# B&R Automation Studio project TD52 (part 33)

### Module_ChargingUnit.var - Module global variables
```iecst
VAR
	bAMM_DPr_AirFilt_A_Hi : BOOL := FALSE; (*Warning charge air filter difference pressure high A*) (*V04.04.00.00*)
	bAMM_DPr_AirFilt_A_Lo : BOOL := FALSE; (*Warning charge air filter difference pressure low A*) (*V04.04.00.00*)
	bAMM_DPr_AirFilt_A_Ms : BOOL := FALSE; (*Warning measurement signal -  charge air filter difference pressure A*)
	bAMM_DPr_AirFilt_B_Hi : BOOL := FALSE; (*Warning charge air filter difference pressure high B*) (*V04.04.00.00*)
	bAMM_DPr_AirFilt_B_Lo : BOOL := FALSE; (*Warning charge air filter difference pressure low B*) (*V04.04.00.00*)
	bAMM_DPr_AirFilt_B_Ms : BOOL := FALSE; (*Warning measurement signal -  charge air filter difference pressure B*)
	bAMM_DPr_AirFilt_Hi : BOOL := FALSE; (*Warning charge air filter difference pressure high*) (*V04.04.00.00*)
	bAMM_DPr_AirFilt_Lo : BOOL := FALSE; (*Warning charge air filter difference pressure low*) (*V04.04.00.00*)
	bAMM_DPr_AirFilt_Ms : BOOL := FALSE; (*Warning measurement signal -  charge air filter difference pressure*)
	bAMM_DPr_Ch_FA_Hi : BOOL := FALSE; (*Warning difference pressure over flame arrester maximum*) (*V04.04.00.00*)
	bAMM_DPr_Ch_HPCooler_Hi : BOOL := FALSE; (*Warning difference pressure over high pressure charge cooler maximum*) (*V04.04.00.00*)
	bAMM_DPr_Ch_LPCooler_Hi : BOOL := FALSE; (*Warning difference pressure over  low pressure charge cooler maximum*) (*V04.04.00.00*)
	bAMM_DPr_Ch_P2s_Hi : BOOL := FALSE; (*Warning charge pressure p2' deviation maximum*) (*V04.07.00.00*)
	bAMM_DPr_Ch_P2s_HiHi : BOOL := FALSE; (*Error charge pressure p2' deviation maximum*)
	bAMM_DPr_Ch_P2_Hi : BOOL := FALSE; (*Warning charge pressure p2 deviation maximum*)
	bAMM_N_TCHP_A_Ms : BOOL := FALSE; (*Warning measurement signal - High pressure turbocharger speed A *)
	bAMM_N_TCHP_B_Ms : BOOL := FALSE; (*Warning measurement signal - High pressure turbocharger speed B*)
	bAMM_N_TCHP_Diff_Hi : BOOL := FALSE; (*Warning High pressure turbocharger speed deviation maximum*)
	bAMM_N_TCHP_Diff_HiHi : BOOL := FALSE; (*Error High pressure turbocharger speed deviation maximum*)
	bAMM_N_TCHP_Hi : BOOL := FALSE; (*Warning High pressure turbocharger speed maximum*)
	bAMM_N_TCHP_HiHi : BOOL := FALSE; (*Error High pressure turbocharger speed maximum*)
	bAMM_N_TCHP_Ms : BOOL := FALSE; (*Warning measurement signal - High pressure turbocharger speed *)
	bAMM_N_TCHP_MsMs : BOOL := FALSE; (*Error measurement signal - BOTH High pressure turbocharger speed *) (*V04.05.01.00*)
	bAMM_N_TCLP_A_Ms : BOOL := FALSE; (*Warning measurement signal - Low pressure turbocharger speed A *)
	bAMM_N_TCLP_B_Ms : BOOL := FALSE; (*Warning measurement signal - Low pressure turbocharger speed B*)
	bAMM_N_TCLP_Diff_Hi : BOOL := FALSE; (*Warning Low pressure turbocharger speed deviation maximum*)
	bAMM_N_TCLP_Diff_HiHi : BOOL := FALSE; (*Error Low pressure turbocharger speed deviation maximum*)
	bAMM_N_TCLP_Hi : BOOL := FALSE; (*Warning Low pressure turbocharger speed maximum*)
	bAMM_N_TCLP_HiHi : BOOL := FALSE; (*Error Low pressure turbocharger speed maximum*)
	bAMM_N_TCLP_Ms : BOOL := FALSE; (*Warning measurement signal - Low pressure turbocharger speed*)
	bAMM_N_TCLP_MsMs : BOOL := FALSE; (*Error measurement signal - BOTH Low pressure turbocharger speed*) (*V04.05.01.00*)
	bAMM_Pr_Ch_OoR : BOOL := FALSE; (*Warning for pressure signals out of range in standstill*)
	bAMM_Pr_Ch_P1HP_A_Ms : BOOL := FALSE; (*Warning measurement signal -  charge pressure p1 before high pressure TC A *)
	bAMM_Pr_Ch_P1HP_B_Ms : BOOL := FALSE; (*Warning measurement signal -  charge pressure p1 before high pressure TC A *)
	bAMM_Pr_Ch_P1HP_Ms : BOOL := FALSE; (*Warning measurement signal -  charge pressure p1 before high pressure TC *)
	bAMM_Pr_Ch_P1LP_A_Ms : BOOL := FALSE; (*Warning measurement signal - charge pressure before  low pressure turbocharger A*) (*V04.04.00.00*)
	bAMM_Pr_Ch_P1LP_B_Ms : BOOL := FALSE; (*Warning measurement signal - charge pressure before  low pressure turbocharger B*) (*V04.04.00.00*)
	bAMM_Pr_Ch_P2bFA_Ms : BOOL := FALSE; (*Warning measurement signal - charge pressure before flame arrester*) (*V04.04.00.00*)
	bAMM_Pr_Ch_P2HP_A_Ms : BOOL := FALSE; (*Warning measurement signal - charge pressure after high pressure turbocharger A*) (*V04.04.00.00*)
	bAMM_Pr_Ch_P2HP_B_Ms : BOOL := FALSE; (*Warning measurement signal - charge pressure after high pressure turbocharger B*) (*V04.04.00.00*)
	bAMM_Pr_Ch_P2HP_Ms : BOOL := FALSE; (*Warning measurement signal - charge pressure after high pressure turbocharger*) (*V04.04.00.00*)
	bAMM_Pr_Ch_P2LP_A_Ms : BOOL := FALSE; (*Warning measurement signal - charge pressure after  low pressure turbocharger A*) (*V04.04.00.00*)
	bAMM_Pr_Ch_P2LP_B_Ms : BOOL := FALSE; (*Warning measurement signal - charge pressure after  low pressure turbocharger B*) (*V04.04.00.00*)
	bAMM_Pr_Ch_P2LP_Ms : BOOL := FALSE; (*Warning measurement signal - charge pressure after  low pressure turbocharger*) (*V04.04.00.00*)
	bAMM_Pr_Ch_P2s_A_Ms : BOOL := FALSE; (*Warning measurement signal -  charge pressure p2' A *)
	bAMM_Pr_Ch_P2s_B_Ms : BOOL := FALSE; (*Warning measurement signal -  charge pressure p2' B*)
	bAMM_Pr_Ch_P2s_MsMs : BOOL := FALSE; (*Error measurement signal -  charge pressure p2' *)
	bAMM_Pr_Ch_P2_A_Ms : BOOL := FALSE; (*Warning measurement signal -  charge pressure p2 A*)
	bAMM_Pr_Ch_P2_B_Ms : BOOL := FALSE; (*Warning measurement signal -  charge pressure p2 B*)
	bAMM_Pr_Ch_P2_MsMs : BOOL := FALSE; (*Error measurement signal -  charge pressure p2 *)
	bAMM_Pr_Ch_P2_Sum_MsMs : BOOL := FALSE; (*Error measurement signal -  sum fault charge pressure *)
	bAMM_T_Ch_T1HP_A_Ms : BOOL := FALSE; (*Warning measurement signal -  charge temperature before high pressure TC  A*) (*V04.05.00.00*)
	bAMM_T_Ch_T1HP_B_Ms : BOOL := FALSE; (*Warning measurement signal -  charge temperature before high pressure TC  B*) (*V04.05.00.00*)
	bAMM_T_Ch_T1HP_Lo : BOOL := FALSE; (*Warning charge temperature before high pressure TC minimum*)
	bAMM_T_Ch_T1HP_MsMs : BOOL := FALSE; (*Error measurement signal -  charge temperature before high pressure TC  *)
	bAMM_T_Ch_T1LP_A_Ms : BOOL := FALSE; (*Warning measurement signal - charge temperature before turbocharger (air intake) A*) (*V04.04.00.00*)
	bAMM_T_Ch_T1LP_B_Ms : BOOL := FALSE; (*Warning measurement signal - charge temperature before turbocharger (air intake) B*) (*V04.04.00.00*)
	bAMM_T_Ch_T1LP_Ms : BOOL := FALSE; (*Warning measurement signal - charge temperature before turbocharger (air intake)*) (*V04.04.00.00*)
	bAMM_T_Ch_T2HP_A_Ms : BOOL := FALSE; (*Warning measurement signal -  charge temperature after high pressure TC  A*) (*V04.05.00.00*)
	bAMM_T_Ch_T2HP_B_Ms : BOOL := FALSE; (*Warning measurement signal -  charge temperature after high pressure TC  B*) (*V04.05.00.00*)
	bAMM_T_Ch_T2HP_HiHi : BOOL := FALSE; (*Error charge temperature after high pressure TC maximum*) (*V04.12.00.00*)
	bAMM_T_Ch_T2HP_Ms : BOOL := FALSE; (*Warning measurement signal -  charge temperature after high pressure TC *) (*V04.05.00.00*)
	bAMM_T_Ch_T2LP_A_Ms : BOOL := FALSE; (*Warning measurement signal -  charge temperature after low pressure TC  A*) (*V04.05.00.00*)
	bAMM_T_Ch_T2LP_B_Ms : BOOL := FALSE; (*Warning measurement signal -  charge temperature after low pressure TC  B*) (*V04.05.00.00*)
	bAMM_T_Ch_T2LP_HiHi : BOOL := FALSE; (*Error charge temperature after low pressure TC maximum*) (*V04.12.00.00*)
	bAMM_T_Ch_T2LP_Ms : BOOL := FALSE; (*Warning measurement signal -  charge temperature after low pressure TC *) (*V04.05.00.00*)
	bAMM_T_Ch_T2s_A_Hi : BOOL := FALSE; (*Warning charge temperature t2' A maximum*)
	bAMM_T_Ch_T2s_A_HiHi : BOOL := FALSE; (*Error charge temperature t2' A maximum*)
	bAMM_T_Ch_T2s_A_Lo : BOOL := FALSE; (*Warning charge temperature t2' A minimum*)
	bAMM_T_Ch_T2s_A_Ms : BOOL := FALSE; (*Warning measurement signal -  charge temperature t2' A*)
	bAMM_T_Ch_T2s_A_RocHiHi : BOOL := FALSE; (*Error charge temperature t2' A rate of change maximum*)
	bAMM_T_Ch_T2s_B_Hi : BOOL := FALSE; (*Warning charge temperature t2' B maximum*)
	bAMM_T_Ch_T2s_B_HiHi : BOOL := FALSE; (*Error charge temperature t2' B maximum*)
	bAMM_T_Ch_T2s_B_Lo : BOOL := FALSE; (*Warning charge temperature t2' B minimum*)
	bAMM_T_Ch_T2s_B_Ms : BOOL := FALSE; (*Warning measurement signal -  charge temperature t2' B*)
	bAMM_T_Ch_T2s_B_RocHiHi : BOOL := FALSE; (*Error charge temperature t2' B rate of change maximum*)
	bAMM_T_Ch_T2s_DiffHi : BOOL := FALSE; (*Warning charge temperature t2' inclination maximum*)
	bAMM_T_Ch_T2s_Hi : BOOL := FALSE; (*Warning charge temperature t2' maximum*)
	bAMM_T_Ch_T2s_HiHi : BOOL := FALSE; (*Error charge temperature t2' maximum*)
	bAMM_T_Ch_T2s_Lo : BOOL := FALSE; (*Warning charge temperature t2' minimum*)
	bAMM_T_Ch_T2s_MsMs : BOOL := FALSE; (*Error measurement signal -  charge temperature t2' *)
	bAMM_T_Ch_T2s_RocHiHi : BOOL := FALSE; (*Error charge temperature t2' rate of change maximum*)
	bAMM_T_Ch_T2_Calc : BOOL := FALSE; (*Warning intercooler inlet temperature not definable*) (*V04.12.00.00*)
	bGCB_On_300s : BOOL := FALSE; (*generator circuit breaker CLOSED + 300s*) (*V04.04.00.00*)
	bGnlTrip : BOOL; (*general alarm trip *)
	bGnlTrip1 : BOOL; (*general alarm trip priority 1*)
	bGnlTrip2 : BOOL; (*general alarm trip priority 2*)
	bGnlTrip3 : BOOL; (*general alarm trip priority 3*)
	bGnlWarning : BOOL; (*general alarm warning *)
	bNetP_Island_20s : BOOL := FALSE; (*Mains parallel operation mode or island mode for 20s*) (*V04.06.00.00*)
	bNoInitDetected : BOOL := FALSE; (*allways true, except 1cycle on init up*)
	bOMSS_MAT : BOOL; (*operation mode selector switch - MANUAL/AUTO/TEST*)
	bP_Nom10_60s : BOOL := FALSE; (*engine power >= 10% of nominal power for 60s*)
	bP_Nom10_300s : BOOL := FALSE; (*engine power >= 10% of nominal power for 300s*)
	bP_Nom10_600s : BOOL := FALSE; (*engine power >= 10% of nominal power for 600s*) (*V04.04.00.00*)
	bP_Nom50_30s : BOOL := FALSE; (*engine power >= 50% of nominal power for 30s*)
	bP_Nom75_02s : BOOL := FALSE; (*engine power >= 75% of nominal power for 2s*) (*V04.04.00.00*)
	bRelModul_ParaSetupOk : BOOL := FALSE; (*Release Module if ParaSetupOk = TRUE*) (*V04.04.00.00*)
	bRelModul_Sys_Run : BOOL := FALSE; (*Release Module if Sys_Run = TRUE*)
	bStartSpd : BOOL := FALSE; (*start speed reached*)
	gastype : INT := 0; (*Actual gas type*)
	iCnt_OpHours_LastCalib : DINT; (*Perm: Actual operating hours at time of calibration*) (*V04.04.00.00*)
	IN_CH : IN_CH_Struct; (*Module IN-Interface*)
	MM2VIS : MM2VIS_Struct; (*Module VISU-Interface (Module --> VISU)*)
	OUT_CH : OUT_CH_Struct; (*Module OUT-Interface*)
	Para : PARA_CH_Struct; (*Module Parameter-Interface*)
	ParaFactoryDefault : PARA_CH_Struct := (0); (*First Init Values*)
	pm : PARA_CH_Struct; (*Stored parameter structure *)
	rNum_Ch_CBV_Valve : REAL := 0.0; (*Number of compressor bypass valve *) (*V04.04.00.00*)
	rP_Act_LastCalib : REAL; (*Perm: Actual electric power at time of calibration [kW]*) (*V04.04.00.00*)
	rT_Ch_T1HP_Max : REAL; (*maximum value - charge temperature before high-pressure TC *) (*V04.05.01.00*)
	rT_Ch_T1LP_Max : REAL; (*maximum value - charge temperature before low-pressure TC *) (*V04.05.01.00*)
	rVol_Ch_AirFilt_Pnom : REAL; (*Perm: Extrapolated value for operation volume flow at nominal power [m³/h]*) (*V04.04.00.00*)
	xEngType : EngType; (*Instance of FB EngType*) (*V04.04.00.00*)
	xOpMode : OpMode := (0); (*Function block for operation mode*)
END_VAR
```

### Program Logical/ChargingUnit/GeneralCH (IEC, version 4.12.0) - general functions

#### GeneralCHCyclic.st - Cyclic code
```iecst
(*******************************************************************************
GeneralCH		general functions

This code is confidential and proprietary to the INNIO Company.
It may not be used in any form, or reproduced in any manner,
without the express written permission of the INNIO Company.
Copyright, INNIO Company, 2019

Customized modifications: -
------------------------

History:
-------
V03.99.00.00	18.03.2013 	Tinello 	Created
V04.04.00.00	18.05.2016 	Tinello 	bP_Nom10_600s added for Spec Vers. c
										Release Module, number of CBV and motor type added
										bP_Nom75_02s, bGCB_On_300s added
V04.06.00.00	01.10.2018 	Tinello 	bNetP_Island_20s added
V04.07.00.00	04.12.2018 	Tinello 	Number of compressor bypass valves added for engine type 4
V04.12.00.00	23.03.2023	Tinello		Added release Sys_Run

(*******************************************************************************)

PROGRAM _CYCLIC

	(* Release Module if ParaSetupOk = TRUE *)
	xTON_ParaSetupOk(IN		:= IN_CH.tPB2MM.bParaSetupOk, PT:= T#10s);
	bRelModul_ParaSetupOk	:= xTON_ParaSetupOk.Q;

	xTON_Sys_Run(IN			:= IN_CH.tPB2MM.bSys_Run, PT:= T#60s);
	bRelModul_Sys_Run		:= xTON_Sys_Run.Q;

	(* Engine motortype *)
	xEngType.Motortype 	:= INT_TO_UINT(Para.iEng_Motortype);
	xEngType();

	(* Operation mode selector switch *)
	bOMSS_MAT 	:= (IN_CH.iIdx_OMSS = 1) OR (IN_CH.iIdx_OMSS = 2) OR (IN_CH.iIdx_OMSS = 3);	(* 1= manual; 2= auto; 3= test mode *)

	(* engine start speed reached *)
	xGR_MAXR_StartSpd(In:= IN_CH.rN_EngAct, Gw := Para.rN_EngStart_LimHi, Hy := Para.rN_EngStart_HyHi);
	xTOF_StartSpd(IN 	:= xGR_MAXR_StartSpd.Q AND bRelModul_ParaSetupOk, PT := T#10s);
	bStartSpd			:= xTOF_StartSpd.Q;

	(* engine power > 10%Pn + 60s / 300s *)
	xGR_MAXR_P_Act10(In := IN_CH.rP_Act_Norm_Filt, Gw:= 0.1, Hy:= 0.01);
	xTON_P_Act10_60(IN	:= xGR_MAXR_P_Act10.Q AND bRelModul_ParaSetupOk AND IN_CH.tGCB_On.Di, PT:= T#60s);
	xTON_P_Act10_300(IN	:= xGR_MAXR_P_Act10.Q AND bRelModul_ParaSetupOk AND IN_CH.tGCB_On.Di, PT:= T#300s);
	xTON_P_Act10_600(IN	:= xGR_MAXR_P_Act10.Q AND bRelModul_ParaSetupOk AND IN_CH.tGCB_On.Di, PT:= T#600s);

	bP_Nom10_60s 		:= xTON_P_Act10_60.Q;
	bP_Nom10_300s 		:= xTON_P_Act10_300.Q;
	bP_Nom10_600s 		:= xTON_P_Act10_600.Q;

	(* engine power > 50%Pn + 30s *)
	xGR_MAXR_P_Act50(In := IN_CH.rP_Act_Norm_Filt, Gw:= 0.5, Hy:= 0.01);
	xTON_P_Act50_30(IN	:= xGR_MAXR_P_Act50.Q AND bRelModul_ParaSetupOk AND IN_CH.tGCB_On.Di, PT:= T#30s);

	bP_Nom50_30s 		:= xTON_P_Act50_30.Q;

	(* engine power > 75%Pn + 2s *)
	xGR_MAXR_P_Act75(In := IN_CH.rP_Act_Norm_Filt, Gw:= 0.75, Hy:= 0.05);
	xTON_P_Act75_02(IN	:= xGR_MAXR_P_Act75.Q AND bRelModul_ParaSetupOk AND IN_CH.tGCB_On.Di, PT:= T#2s);

	bP_Nom75_02s 		:= xTON_P_Act75_02.Q;

	(* generator circuit breaker CLOSED + 300s *)
	xTON_GCB_On_300(IN	:= IN_CH.tGCB_On.Di, PT:= T#300s);
	bGCB_On_300s 		:= xTON_GCB_On_300.Q;

	(* call function for the state machine - engine operation mode *)
	xOpMode(in 	:= IN_CH.iSt_OpMode);

	(* Mains parallel operation mode / island mode + 20s *)
	xTON_NetP_Island_20(IN	:= xOpMode.NetP OR xOpMode.Island, PT:= T#20s);
	bNetP_Island_20s		:= xTON_NetP_Island_20.Q;

	(* gastype *)
	gastype	:= IN_CH.iIdx_Gtyp_Dem;

	(* Number of compressor bypass valves *)
	CASE Para.iEng_Motortype OF
		412:	IF xOpMode.Island						 	THEN	rNum_Ch_CBV_Valve	:= 2;
															ELSE	rNum_Ch_CBV_Valve	:= 1;
				END_IF
		416:	IF xOpMode.Island						 	THEN	rNum_Ch_CBV_Valve	:= 2;
															ELSE	rNum_Ch_CBV_Valve	:= 1;
				END_IF
		420:	IF xOpMode.Island						 	THEN	rNum_Ch_CBV_Valve	:= 2;
															ELSE	rNum_Ch_CBV_Valve	:= 1;
				END_IF
		424:	IF xOpMode.Island						 	THEN	rNum_Ch_CBV_Valve	:= 2;
															ELSE	rNum_Ch_CBV_Valve	:= 1;
				END_IF
		612:														rNum_Ch_CBV_Valve	:= 1;
		616:														rNum_Ch_CBV_Valve	:= 2;
		620:														rNum_Ch_CBV_Valve	:= 3;
		624:	IF FIND(IN_CH.szEng_Motorversion, 'H') = 1 	THEN	rNum_Ch_CBV_Valve	:= 2;
															ELSE	rNum_Ch_CBV_Valve	:= 4;
				END_IF
		920:														rNum_Ch_CBV_Valve	:= 2;
	END_CASE

END_PROGRAM
```

#### GeneralCH.var - Local variables
```iecst
VAR
	xGR_MAXR_P_Act10 : GR_MAXR := (0); (*FuB*)
	xGR_MAXR_P_Act50 : GR_MAXR := (0); (*FuB*)
	xGR_MAXR_P_Act75 : GR_MAXR := (0); (*FuB*)
	xGR_MAXR_StartSpd : GR_MAXR := (0); (*Engine start speed passed*)
	xTOF_StartSpd : TOF := (0); (*FuB*)
	xTON_GCB_On_300 : TON := (0); (*FuB*)
	xTON_NetP_Island_20 : TON := (0); (*FuB*)
	xTON_ParaSetupOk : TON := (0); (*FuB*)
	xTON_P_Act10_60 : TON := (0); (*FuB*)
	xTON_P_Act10_300 : TON := (0); (*FuB*)
	xTON_P_Act10_600 : TON := (0); (*FuB*)
	xTON_P_Act50_30 : TON := (0); (*FuB*)
	xTON_P_Act75_02 : TON := (0); (*FuB*)
	xTON_Sys_Run : TON := (0); (*FuB*)
END_VAR
```

### Program Logical/ChargingUnit/DefaultCH (IEC, version 4.00.0) - Settings default values

#### DefaultCHCyclic.st - Cyclic code
```iecst
(*******************************************************************************
DefaultCH		value set

This code is confidential and proprietary to the INNIO Company.
It may not be used in any form, or reproduced in any manner,
without the express written permission of the INNIO Company.
Copyright, INNIO Company, 2019

Customized modifications: -
------------------------

History:
-------
V03.99.00.00	11.09.2012	Tinello		new

Instructions for use:
--------------------
- Default TRUE setting for not existing Di's

Outstandings:
------------

*******************************************************************************)
PROGRAM _CYCLIC

END_PROGRAM
```

### Program Logical/ChargingUnit/CH_SpeedTC (IEC, version 4.12.0) - turbo charger speed

#### CH_SpeedTCCyclic.st - Cyclic code
```iecst
(*******************************************************************************
TC_Speed	 		 turbocharger speed

This code is confidential and proprietary to the INNIO Company.
It may not be used in any form, or reproduced in any manner,
without written permission of the INNIO Company.
Copyright, INNIO Company, 2023

- turbocharger speed measuring
- speed and signal monitoring
- power reduction

Customized modifications: -
------------------------

History:
-------
V03.99.00.00	18.03.2013	Tinello		restructured
V04.00.00.00	01.09.2014	Tinello		If engine speed = 0 and no measurement failure -> TC speed is set to 0
V04.04.00.00	27.10.2016	Tinello		change of speed deviation function -> Spec.(b)
V04.05.00.00	23.01.2018	Tinello		Release Monitoring hinzu und Warnmanagement vereinfacht
V04.05.01.00	15.03.2018	Tinello		Spezifikation c
V04.05.03.00	28.05.2018	Tinello		Bugfix: Quittierung der Ms-Sto
V04.07.00.00	13.06.2019	Tinello		MsErr active with op.switch OFF mode / interpolated speed max limit -> Spezifikation d
V04.10.00.00	26.01.2021	Tinello		2x out-interface for interpolated TC speed max limit / Use intake air temperature if T1HP is not available
										BugFix: Timer-FuB's
V04.12.00.00	17.01.2023 	Tinello		Extrapolation of TC speed limit
V04.14.00.00	18.03.2025	Theobald	Alarm 2325, 2326 and 2327 only appear when there is too low TC speed and the TC speed sensor is in good quality.

(*******************************************************************************)
PROGRAM _CYCLIC

	xTON_1000ms(IN:= NOT xTON_1000ms.Q, PT:= T#800ms);											(* 800ms + 2x cycle time = 1000 ms *)

	(*------------------------------------------------------*)
	(* RESET of alarms and warnings 						*)
	(*------------------------------------------------------*)
	bAMM_N_TCLP_Ms			:= FALSE;
	bAMM_N_TCLP_MsMs		:= FALSE;
	bAMM_N_TCLP_A_Ms 		:= FALSE;
	bAMM_N_TCLP_B_Ms 		:= FALSE;
	bAMM_N_TCLP_Hi			:= FALSE;
	bAMM_N_TCLP_HiHi		:= FALSE;
	bAMM_N_TCLP_Diff_Hi		:= FALSE;
	bAMM_N_TCLP_Diff_HiHi	:= FALSE;

	bAMM_N_TCHP_Ms			:= FALSE;
	bAMM_N_TCHP_MsMs		:= FALSE;
	bAMM_N_TCHP_A_Ms 		:= FALSE;
	bAMM_N_TCHP_B_Ms 		:= FALSE;
	bAMM_N_TCHP_Hi			:= FALSE;
	bAMM_N_TCHP_HiHi		:= FALSE;
	bAMM_N_TCHP_Diff_Hi		:= FALSE;
	bAMM_N_TCHP_Diff_HiHi	:= FALSE;

	OUT_CH.rP_Red_TC_Norm 	:= 1;																(* release full load -> no reduction *)
	OUT_CH.rN_TCLP_HiHi		:= Para.rN_TCLP_HiHi;
	OUT_CH.rN_TCHP_HiHi		:= Para.rN_TCHP_HiHi;

	(*------------------------------------------------------*)
	(* VISU var of module									*)
	(*------------------------------------------------------*)
	(* In case of no engine speed and no measurement failure -> TC speed is set to 0 *)
	IF IN_CH.rN_EngAct > 10 OR (IN_CH.tN_TCLP.Ai   > 5000) OR (IN_CH.tN_TCLP.Ai   < -5000) 	THEN
		MM2VIS.rN_TCLP		:= IN_CH.tN_TCLP.Ai;
	ELSE
		MM2VIS.rN_TCLP		:= 0;
	END_IF

	IF IN_CH.rN_EngAct > 10 OR (IN_CH.tN_TCLP_A.Ai > 5000) OR (IN_CH.tN_TCLP_A.Ai < -5000)	THEN
		MM2VIS.rN_TCLP_A	:= IN_CH.tN_TCLP_A.Ai;
	ELSE
		MM2VIS.rN_TCLP_A	:= 0;
	END_IF

	IF IN_CH.rN_EngAct > 10 OR (IN_CH.tN_TCLP_B.Ai > 5000) OR (IN_CH.tN_TCLP_B.Ai < -5000)	THEN
		MM2VIS.rN_TCLP_B	:= IN_CH.tN_TCLP_B.Ai;
	ELSE
		MM2VIS.rN_TCLP_B	:= 0;
	END_IF

	IF IN_CH.rN_EngAct > 10 OR (IN_CH.tN_TCHP.Ai   > 5000) OR (IN_CH.tN_TCHP.Ai   < -5000)  THEN
		MM2VIS.rN_TCHP		:= IN_CH.tN_TCHP.Ai;
	ELSE
		MM2VIS.rN_TCHP		:= 0;
	END_IF

	IF IN_CH.rN_EngAct > 10 OR (IN_CH.tN_TCHP_A.Ai > 5000) OR (IN_CH.tN_TCHP_A.Ai < -5000)	THEN
		MM2VIS.rN_TCHP_A	:= IN_CH.tN_TCHP_A.Ai;
	ELSE
		MM2VIS.rN_TCHP_A	:= 0;
	END_IF

	IF IN_CH.rN_EngAct > 10 OR (IN_CH.tN_TCHP_B.Ai > 5000) OR (IN_CH.tN_TCHP_B.Ai < -5000)	THEN
		MM2VIS.rN_TCHP_B	:= IN_CH.tN_TCHP_B.Ai;
	ELSE
		MM2VIS.rN_TCHP_B	:= 0;
	END_IF

	(*------------------------------------------------------*)
	(* check if any turbocharger speed measuring is active 	*)
	(*------------------------------------------------------*)
	IF 	(Para.bN_TCHP_Exist OR Para.bN_TCHP_A_Exist OR Para.bN_TCHP_B_Exist OR					(* High pressure turbocharger exist *)
		 Para.bN_TCLP_Exist OR Para.bN_TCLP_A_Exist OR Para.bN_TCLP_B_Exist	  ) AND				(* Low  pressure turbocharger exist *)
		bRelModul_ParaSetupOk AND IN_CH.tPB2MM.bSys_Run
	THEN
		(*--------------------------------------------------*)
		(* measurement signal failure or signal too low		*)
		(*--------------------------------------------------*)
			(* Check if signal is too low --> TC speed < 60% of TC speed maximum and actual Power > 95% *)
			bN_TCLP_ErrMsLow		:= (IN_CH.tN_TCLP.Ai   < (Para.rN_TCLP_HiHi * 0.6)) AND (IN_CH.rP_Act_Norm_Filt > 0.95);
			bN_TCLP_A_ErrMsLow		:= (IN_CH.tN_TCLP_A.Ai < (Para.rN_TCLP_HiHi * 0.6)) AND (IN_CH.rP_Act_Norm_Filt > 0.95);
			bN_TCLP_B_ErrMsLow		:= (IN_CH.tN_TCLP_B.Ai < (Para.rN_TCLP_HiHi * 0.6)) AND (IN_CH.rP_Act_Norm_Filt > 0.95);

			bN_TCHP_ErrMsLow		:= (IN_CH.tN_TCHP.Ai   < (Para.rN_TCHP_HiHi * 0.6)) AND (IN_CH.rP_Act_Norm_Filt > 0.95);
			bN_TCHP_A_ErrMsLow		:= (IN_CH.tN_TCHP_A.Ai < (Para.rN_TCHP_HiHi * 0.6)) AND (IN_CH.rP_Act_Norm_Filt > 0.95);
			bN_TCHP_B_ErrMsLow		:= (IN_CH.tN_TCHP_B.Ai < (Para.rN_TCHP_HiHi * 0.6)) AND (IN_CH.rP_Act_Norm_Filt > 0.95);

		(* Low pressure turbocharger speed *)
		bAMM_N_TCLP_Ms 				:= (bN_TCLP_ErrMsLow   OR NOT IN_CH.tN_TCLP.GoodQual) 	AND Para.bN_TCLP_Exist;							(* W2617 *)
		bAMM_N_TCLP_A_Ms 			:= (bN_TCLP_A_ErrMsLow OR NOT IN_CH.tN_TCLP_A.GoodQual) AND Para.bN_TCLP_A_Exist;						(* W2565 *)
		bAMM_N_TCLP_B_Ms 			:= (bN_TCLP_B_ErrMsLow OR NOT IN_CH.tN_TCLP_B.GoodQual) AND Para.bN_TCLP_B_Exist;						(* W2566 *)
		bAMM_N_TCLP_MsMs			:=  bAMM_N_TCLP_A_Ms AND bAMM_N_TCLP_B_Ms AND IN_CH.tN_TCLP_A.GoodQual AND IN_CH.tN_TCLP_B.GoodQual;	(* A2327 *)

		(* turbocharger speed *)
		bAMM_N_TCHP_Ms				:= (bN_TCHP_ErrMsLow   OR NOT IN_CH.tN_TCHP.GoodQual) 	AND Para.bN_TCHP_Exist;							(* W2615 *)	(* W2616 *)
		bAMM_N_TCHP_A_Ms			:= (bN_TCHP_A_ErrMsLow OR NOT IN_CH.tN_TCHP_A.GoodQual) AND Para.bN_TCHP_A_Exist;						(* W3522 *)	(* W2563 *)
		bAMM_N_TCHP_B_Ms			:= (bN_TCHP_B_ErrMsLow OR NOT IN_CH.tN_TCHP_B.GoodQual) AND Para.bN_TCHP_B_Exist;						(* W3523 *)	(* W2564 *)
		bAMM_N_TCHP_MsMs			:=  bAMM_N_TCHP_A_Ms AND bAMM_N_TCHP_B_Ms AND IN_CH.tN_TCHP_A.GoodQual AND IN_CH.tN_TCHP_B.GoodQual;	(* A2325 *)	(* A2326 *)

			(* release monitoring	*)
			xTON_RelMon_N_TCLP(IN	:= Para.bN_TCLP_Exist   AND NOT bAMM_N_TCLP_Ms,   PT:= T#10s);
			xTON_RelMon_N_TCLP_A(IN	:= Para.bN_TCLP_A_Exist AND NOT bAMM_N_TCLP_A_Ms, PT:= T#10s);
			xTON_RelMon_N_TCLP_B(IN	:= Para.bN_TCLP_B_Exist AND NOT bAMM_N_TCLP_B_Ms, PT:= T#10s);

			xTON_RelMon_N_TCHP(IN	:= Para.bN_TCHP_Exist   AND NOT bAMM_N_TCHP_Ms,   PT:= T#10s);
			xTON_RelMon_N_TCHP_A(IN	:= Para.bN_TCHP_A_Exist AND NOT bAMM_N_TCHP_A_Ms, PT:= T#10s);
			xTON_RelMon_N_TCHP_B(IN	:= Para.bN_TCHP_B_Exist AND NOT bAMM_N_TCHP_B_Ms, PT:= T#10s);

			bRelMon_N_TCLP			:= xTON_RelMon_N_TCLP.Q;
			bRelMon_N_TCLP_A		:= xTON_RelMon_N_TCLP_A.Q;
			bRelMon_N_TCLP_B		:= xTON_RelMon_N_TCLP_B.Q;

			bRelMon_N_TCHP			:= xTON_RelMon_N_TCHP.Q;
			bRelMon_N_TCHP_A		:= xTON_RelMon_N_TCHP_A.Q;
			bRelMon_N_TCHP_B		:= xTON_RelMon_N_TCHP_B.Q;

		IF	bP_Nom10_60s THEN
			(*--------------------------------------------------*)
			(* turbocharger speed MAX 					  		*)
			(*--------------------------------------------------*)

			(* At least one low-pressure turbocharger speed > interpolated speed limit or max limit *)
				rN_TCLP_Max				:= MAX(IN_CH.tN_TCLP.Ai   * BOOL_TO_REAL(bRelMon_N_TCLP),
										 	   IN_CH.tN_TCLP_A.Ai * BOOL_TO_REAL(bRelMon_N_TCLP_A),
											   IN_CH.tN_TCLP_B.Ai * BOOL_TO_REAL(bRelMon_N_TCLP_B));

				xLCRScal_N_TCLP_Hi(x	:= rT_Ch_T1LP_Max,									(* inter- and extrapolation of allowed TC speed  *)
								   x1	:= Para.rT_Ch_T1LP_Hi,								(* depending on the inlet temperature *)
								   x2	:= Para.rT_Ch_T1LP_HiHi,
								   y1	:= Para.rN_TCLP_TempLimit_HiHi,
								   y2	:= Para.rN_TCLP_TempLimit_Hi);

				xLCRScal_N_TCLP_HiHi(x	:= rT_Ch_T1LP_Max,									(* inter- and extrapolation of allowed TC MAX speed  *)
								     x1	:= Para.rT_Ch_T1LP_Hi,								(* depending on the inlet temperature *)
								 	 x2	:= Para.rT_Ch_T1LP_HiHi,
									 y1	:= Para.rN_TCLP_HiHi,
									 y2	:= Para.rN_TCLP_Hi);

			bAMM_N_TCLP_DB				:= rN_TCLP_Max > LIMIT(0, xLCRScal_N_TCLP_Hi.y,   Para.rN_TCLP_TempLimit_HiHi) * 0.99;	(* deadband *)
			bAMM_N_TCLP_Hi				:= rN_TCLP_Max > LIMIT(0, xLCRScal_N_TCLP_Hi.y,   Para.rN_TCLP_TempLimit_HiHi);			(* -> power reduction *)(* W2527 *)
			bAMM_N_TCLP_HiHi			:= rN_TCLP_Max > LIMIT(0, xLCRScal_N_TCLP_HiHi.y, Para.rN_TCLP_HiHi);											(* A2239 *)

			OUT_CH.rN_TCLP_HiHi			:= LIMIT(0, xLCRScal_N_TCLP_HiHi.y, Para.rN_TCLP_HiHi);

			(* At least one high-pressure turbocharger speed > interpolated speed limit or max limit *)
				rN_TCHP_Max				:= MAX(IN_CH.tN_TCHP.Ai   * BOOL_TO_REAL(bRelMon_N_TCHP),
											   IN_CH.tN_TCHP_A.Ai * BOOL_TO_REAL(bRelMon_N_TCHP_A),
											   IN_CH.tN_TCHP_B.Ai * BOOL_TO_REAL(bRelMon_N_TCHP_B));

				xLCRScal_N_TCHP_Hi(  x	:= rT_Ch_T1HP_Max,									(* inter- and extrapolation of allowed TC speed  *)
								  	 x1	:= Para.rT_Ch_T1HP_Hi,								(* depending on the inlet temperature *)
								  	 x2	:= Para.rT_Ch_T1HP_HiHi,
								  	 y1	:= Para.rN_TCHP_TempLimit_HiHi,
								  	 y2	:= Para.rN_TCHP_TempLimit_Hi);

				xLCRScal_N_TCHP_HiHi(x	:= rT_Ch_T1HP_Max,									(* inter- and extrapolation of allowed TC speed  *)
									 x1	:= Para.rT_Ch_T1HP_Hi,								(* depending on the inlet temperature *)
								  	 x2	:= Para.rT_Ch_T1HP_HiHi,
								  	 y1	:= Para.rN_TCHP_HiHi,
								  	 y2	:= Para.rN_TCHP_Hi);

			bAMM_N_TCHP_DB				:= rN_TCHP_Max > LIMIT(0, xLCRScal_N_TCHP_Hi.y,   Para.rN_TCHP_TempLimit_HiHi) * 0.996;	(* deadband *)
			bAMM_N_TCHP_Hi				:= rN_TCHP_Max > LIMIT(0, xLCRScal_N_TCHP_Hi.y,   Para.rN_TCHP_TempLimit_HiHi);			(* -> power reduction*)	(* W3524 *)	(* W2526 *)
			bAMM_N_TCHP_HiHi			:= rN_TCHP_Max > LIMIT(0, xLCRScal_N_TCHP_HiHi.y, Para.rN_TCHP_HiHi);											(* A2278 *)	(* A2237 *)

			OUT_CH.rN_TCHP_HiHi			:= LIMIT(0, xLCRScal_N_TCHP_HiHi.y, Para.rN_TCHP_HiHi);

			(*--------------------------------------------------*)
			(* turbocharger speed deviation (Spreizung)			*)
			(*--------------------------------------------------*)
			IF 	bRelMon_N_TCHP_A AND bRelMon_N_TCHP_B
			THEN
				bAMM_N_TCHP_Diff_Hi		:= ABS(IN_CH.tN_TCHP_A.Ai - IN_CH.tN_TCHP_B.Ai) > Para.rN_TC_Diff_Hi;			(* W2614 *)	(* W2528 *)
				bAMM_N_TCHP_Diff_HiHi	:= ABS(IN_CH.tN_TCHP_A.Ai - IN_CH.tN_TCHP_B.Ai) > Para.rN_TC_Diff_Hi + 400;		(* A2279 *)	(* A2225 *)
			END_IF

			IF 	bRelMon_N_TCLP_A AND bRelMon_N_TCLP_B
			THEN
				bAMM_N_TCLP_Diff_Hi		:= ABS(IN_CH.tN_TCLP_A.Ai - IN_CH.tN_TCLP_B.Ai) > Para.rN_TC_Diff_Hi;						(* W2529 *)
				bAMM_N_TCLP_Diff_HiHi	:= ABS(IN_CH.tN_TCLP_A.Ai - IN_CH.tN_TCLP_B.Ai) > Para.rN_TC_Diff_Hi + 400;					(* A2226 *)
			END_IF

			(*--------------------------------------------------*)
			(* POWER REDUCTION and LIMITATION					*)																	(* B2144 *)
			(*--------------------------------------------------*)

			(* reduction by speed maximum 	*)
			IF xTON_1000ms.Q THEN																(* check every second *)

				IF 		   bAMM_N_TCHP_Hi OR bAMM_N_TCLP_Hi  THEN 	iTi_N_TC_P_Red_dur 			:= iTi_N_TC_P_Red_dur 	    + 1;
																	iTi_N_TC_P_Red_reset_dur	:= 0;
				ELSIF NOT (bAMM_N_TCHP_DB OR bAMM_N_TCLP_DB)
					  AND rP_Red_N_TC_Max < 1		 		 THEN 	iTi_N_TC_P_Red_dur 			:= 0;
																	iTi_N_TC_P_Red_reset_dur	:= iTi_N_TC_P_Red_reset_dur + 1;
				ELSE
																	iTi_N_TC_P_Red_dur 			:= 0;
																	iTi_N_TC_P_Red_reset_dur	:= 0;
				END_IF
			END_IF

			IF iTi_N_TC_P_Red_dur >= 120 THEN
				bAMM_N_TCHP_HiHi	:= bAMM_N_TCHP_HiHi OR bAMM_N_TCHP_Hi;												(* A2278 *)	(* A2237 *)
				bAMM_N_TCLP_HiHi	:= bAMM_N_TCLP_HiHi OR bAMM_N_TCLP_Hi;															(* A2239 *)
			END_IF

			xTON_P_Red_TC_MaxInc(IN:= iTi_N_TC_P_Red_dur 	   > 0 AND NOT xTON_P_Red_TC_MaxInc.Q, PT:= T#30s);
			xTON_P_Red_TC_MaxDec(IN:= iTi_N_TC_P_Red_reset_dur > 0 AND NOT xTON_P_Red_TC_MaxDec.Q, PT:= T#30s);

			IF EDGEPOS(iTi_N_TC_P_Red_dur > 0) THEN	rP_Red_N_TC_Max	:= LIMIT(0.5, rP_Act_Norm_Save1 - Para.rP_Red_TC, 		1);	END_IF
			IF EDGEPOS(xTON_P_Red_TC_MaxInc.Q) THEN	rP_Red_N_TC_Max	:= LIMIT(0.5, rP_Red_N_TC_Max 	- Para.rP_Red_TC, 		1);	END_IF
			IF EDGEPOS(xTON_P_Red_TC_MaxDec.Q) THEN	rP_Red_N_TC_Max	:= LIMIT(0.5, rP_Red_N_TC_Max 	+ Para.rP_Red_TC_reset, 1);	END_IF

			IF iTi_N_TC_P_Red_dur = 0 THEN
				rP_Act_Norm_Save1	:= IN_CH.rP_Act_Norm_Filt;									(* save actual power *)
			END_IF

			OUT_CH.rP_Red_TC_Norm 	:= MIN(OUT_CH.rP_Red_TC_Norm, rP_Red_N_TC_Max);				(* Power reduction *)

			(* reduction by speed deviation - until user acknowledge *)
			IF 	MM2VIS.bMsg2614 OR																(*  			 TC speed deviation maximum *)
				MM2VIS.bMsg2528 OR																(* High pressure TC speed deviation maximum *)
				MM2VIS.bMsg2529																	(*  Low pressure TC speed deviation maximum *)
			THEN
				rP_Red_N_TC_Diff		:= LIMIT(0.5, rP_Act_Norm_Save - Para.rP_Red_TC, 1);	(* reduction start from actual power *)
				OUT_CH.rP_Red_TC_Norm 	:= MIN(OUT_CH.rP_Red_TC_Norm, rP_Red_N_TC_Diff);
			ELSE
				rP_Act_Norm_Save		:= IN_CH.rP_Act_Norm_Filt;								(* save actual power *)
			END_IF

			(* power limitation by signal failure or signal too low error *)
			xTON_P_Red_TC_Ms(IN	:= bAMM_N_TCHP_Ms OR bAMM_N_TCHP_A_Ms OR bAMM_N_TCHP_B_Ms OR
								   bAMM_N_TCLP_Ms OR bAMM_N_TCLP_A_Ms OR bAMM_N_TCLP_B_Ms,
							 PT	:= T#10s);

			IF xTON_P_Red_TC_Ms.Q THEN
				OUT_CH.rP_Red_TC_Norm 	:= MIN(OUT_CH.rP_Red_TC_Norm, 0.7);						(* power-LIMITATION to 70% P nominal *)
			END_IF

		ELSE
			(* reset power reduction *)
			iTi_N_TC_P_Red_dur			:= 0;
			iTi_N_TC_P_Red_reset_dur	:= 0;
			rP_Red_N_TC_Max				:= 1;													(* release full load -> no reduction *)

			(* save actual power *)
			rP_Act_Norm_Save			:= IN_CH.rP_Act_Norm_Filt;
			rP_Act_Norm_Save1			:= IN_CH.rP_Act_Norm_Filt;

			(* reset timer *)
			xTON_P_Red_TC_MaxInc(IN		:= FALSE);
			xTON_P_Red_TC_MaxDec(IN		:= FALSE);
			xTON_P_Red_TC_Ms(IN			:= FALSE);
		END_IF
	ELSE
		(* reset power reduction *)
		iTi_N_TC_P_Red_dur				:= 0;
		iTi_N_TC_P_Red_reset_dur		:= 0;
		rP_Red_N_TC_Max					:= 1;													(* release full load -> no reduction *)

		(* save actual power *)
		rP_Act_Norm_Save				:= IN_CH.rP_Act_Norm_Filt;
		rP_Act_Norm_Save1				:= IN_CH.rP_Act_Norm_Filt;

		(* reset timer/release monitoring *)
		xTON_RelMon_N_TCLP(IN			:= FALSE);
		xTON_RelMon_N_TCLP_A(IN			:= FALSE);
		xTON_RelMon_N_TCLP_B(IN			:= FALSE);
		xTON_RelMon_N_TCHP(IN			:= FALSE);
		xTON_RelMon_N_TCHP_A(IN			:= FALSE);
		xTON_RelMon_N_TCHP_B(IN			:= FALSE);
		xTON_P_Red_TC_MaxInc(IN			:= FALSE);
		xTON_P_Red_TC_MaxDec(IN			:= FALSE);
		xTON_P_Red_TC_Ms(IN				:= FALSE);
		bRelMon_N_TCLP					:= FALSE;
		bRelMon_N_TCLP_A				:= FALSE;
		bRelMon_N_TCLP_B				:= FALSE;
		bRelMon_N_TCHP					:= FALSE;
		bRelMon_N_TCHP_A				:= FALSE;
		bRelMon_N_TCHP_B				:= FALSE;
	END_IF

END_PROGRAM
```

#### CH_SpeedTC.var - Local variables
```iecst
VAR
	bAMM_N_TCHP_DB : BOOL := 0; (*High pressure turbocharger speed higher than deadband limit*)
	bAMM_N_TCLP_DB : BOOL := 0; (*Low pressure turbocharger speed higher than deadband limit*)
	bN_TCHP_A_ErrMsLow : BOOL := FALSE; (*ERROR - High pressure turbocharger speed A signal -  too low *)
	bN_TCHP_B_ErrMsLow : BOOL := FALSE; (*ERROR - High pressure turbocharger speed B signal -  too low *)
	bN_TCHP_ErrMsLow : BOOL := FALSE; (*ERROR - High pressure turbocharger speed signal -  too low *)
	bN_TCLP_A_ErrMsLow : BOOL := FALSE; (*ERROR - Low pressure turbocharger speed A signal -  too low *)
	bN_TCLP_B_ErrMsLow : BOOL := FALSE; (*ERROR - Low pressure turbocharger speed B signal -  too low *)
	bN_TCLP_ErrMsLow : BOOL := FALSE; (*ERROR - Low pressure turbocharger speed signal -  too low *)
	bRelMon_N_TCHP : BOOL := FALSE; (*Release monitoring high-pressure turbocharger speed*)
	bRelMon_N_TCHP_A : BOOL := FALSE; (*Release monitoring high-pressure turbocharger speed A*)
	bRelMon_N_TCHP_B : BOOL := FALSE; (*Release monitoring high-pressure turbocharger speed B*)
	bRelMon_N_TCLP : BOOL := FALSE; (*Release monitoring low-pressure turbocharger speed*)
	bRelMon_N_TCLP_A : BOOL := FALSE; (*Release monitoring low-pressure turbocharger speed A*)
	bRelMon_N_TCLP_B : BOOL := FALSE; (*Release monitoring low-pressure turbocharger speed B*)
	iTi_N_TC_P_Red_dur : UDINT := 0; (*Timer - time of power reduction by charge temperature before HP TC maximum [s]*)
	iTi_N_TC_P_Red_reset_dur : UDINT := 0; (*Timer - time of power reduction by charge temperature before HP TC maximum [s]*)
	rN_TCHP_Max : REAL := 0; (*maximum value - high-pressure turbocharger speed [rpm]*)
	rN_TCLP_Max : REAL := 0; (*maximum value - low-pressure turbocharger speed [rpm]*)
	rP_Act_Norm_Save : REAL := 0.0; (*Save actual power for power reduction by TC [%Pnom]*)
	rP_Act_Norm_Save1 : REAL := 0.0; (*Save actual power for power reduction by TC [%Pnom]*)
	rP_Red_N_TC_Diff : REAL := 1; (*power reduction by turbocharger speed deviation*)
	rP_Red_N_TC_Max : REAL := 1; (*power reduction by turbocharger speed maximum*)
	xLCRScal_N_TCHP_Hi : LCRScal := (0); (*FuB*)
	xLCRScal_N_TCHP_HiHi : LCRScal := (0); (*FuB*)
	xLCRScal_N_TCLP_Hi : LCRScal := (0); (*FuB*)
	xLCRScal_N_TCLP_HiHi : LCRScal := (0); (*FuB*)
	xTON_1000ms : TON := (0); (*FuB*)
	xTON_P_Red_TC_MaxDec : TON := (0); (*FuB*)
	xTON_P_Red_TC_MaxInc : TON := (0); (*FuB*)
	xTON_P_Red_TC_Ms : TON := (0); (*FuB*)
	xTON_RelMon_N_TCHP : TON := (0); (*FuB*)
	xTON_RelMon_N_TCHP_A : TON := (0); (*FuB*)
	xTON_RelMon_N_TCHP_B : TON := (0); (*FuB*)
	xTON_RelMon_N_TCLP : TON := (0); (*FuB*)
	xTON_RelMon_N_TCLP_A : TON := (0); (*FuB*)
	xTON_RelMon_N_TCLP_B : TON := (0); (*FuB*)
END_VAR
```

### Program Logical/ChargingUnit/CH_Temp (IEC, version 4.12.0) - charging temperature

#### CH_TempCyclic.st - Cyclic code
```iecst
(*******************************************************************************
CH_Temp	 			 Charging temperatures

This code is confidential and proprietary to the INNIO Company.
It may not be used in any form, or reproduced in any manner,
without written permission of the INNIO Company.
Copyright, INNIO Company, 2023

Customized modifications: -
------------------------

History:
-------
V03.99.00.00	30.11.2012	Tinello		restructured
V04.01.00.00	19.05.2014	Tinello		gastype = 0 included
				02.06.2014	Tinello 	bugfix power reduction
				07.08.2014	Tinello		Changed activation of charge temperature maximum monitoring
V04.04.00.00	18.05.2016 	Tinello 	bP_Nom10_600s added --> Spec Vers. c
				02.11.2016 	Tinello		T1LP and monitoring added --> Spec Vers. c
				25.01.2017	Tinello		bugfix for AVG
V04.05.00.00	06.02.2017	Tinello		vvm cycle time correction
				19.04.2017	Weitzer		2460, 2461 added, SWAT920/2
										2221, 2222 modified, SWAT920/2
										2223 incl. P reduction modified, SWAT920/2
				27.04.2017	lettenb.	920: set OUT_CH.rT_Ch_T2s_x to Para.rT_Ch_T2s_Hi[gastype] in case of MS_A + MS_B, SWAT920/2
V04.05.01.00	10.10.2017	Zingerle	Spezifikation f komplett eingearbeitet und abgeglichen
				24.01.2018	Tinello		Cleanup and final modifications
V04.05.02.00	15.03.2018	Tinello		BugFix --> Anzeige Temp bei BWS aus
V04.05.03.00	19.03.2018	Tinello		Spezifikation g
V04.06.00.00	26.09.2018	Perktold	20s delay after SY until activation of T2s max monitoring - Spezifikation h
V04.07.00.00	15.05.2019	Tinello		Spezifikation i: MsErr active with op.switch OFF mode / Handover T1 before HP TC TO other modules
														 No warning	if speed sensors available
V04.12.00.00	24.04.2023 	Tinello		Deleted T1 maximum monitoring / Added calculation, monitoring and power red of T2 max

(*******************************************************************************)
PROGRAM _INIT
	(* ramp settings *)
	xRAMPE_R_P_Red_Ch_T2LP.TC_Time	:= TASK_TIME_10MS;
	xRAMPE_R_P_Red_Ch_T2LP.Rise		:= 0.001;		(*  0,1% Pnom/s *)
	xRAMPE_R_P_Red_Ch_T2LP.Sink		:= 0.1;			(* 10,0% Pnom/s *)

	xRAMPE_R_P_Red_Ch_T2HP.TC_Time	:= TASK_TIME_10MS;
	xRAMPE_R_P_Red_Ch_T2HP.Rise		:= 0.001;		(*  0,1% Pnom/s *)
	xRAMPE_R_P_Red_Ch_T2HP.Sink		:= 0.1;			(* 10,0% Pnom/s *)

END_PROGRAM

PROGRAM _CYCLIC

	(*--------------------------------------------------*)
	(* RESET of alarms and warnings 					*)
	(*--------------------------------------------------*)
	xTON_200msTick(IN	:= NOT xTON_200msTick.Q, PT:= T#180ms);							(* 180ms + 2x cycle time = 200 ms *)

	IF xTON_200msTick.Q THEN															(* to notice the alarm in 100ms Task *)

		bAMM_T_Ch_T1LP_Ms		:= FALSE;		(* W2411 *)
		bAMM_T_Ch_T1LP_A_Ms		:= FALSE;		(* W2413 *)
		bAMM_T_Ch_T1LP_B_Ms		:= FALSE;		(* W2414 *)

		bAMM_T_Ch_T2LP_Ms		:= FALSE;		(* W2489 *)
		bAMM_T_Ch_T2LP_A_Ms		:= FALSE;		(* W2481 *)
		bAMM_T_Ch_T2LP_B_Ms		:= FALSE;		(* W2482 *)
		bAMM_T_Ch_T2LP_HiHi		:= FALSE;		(* A2370 *)
		bAMM_T_Ch_T2_Calc		:= FALSE;		(* W9370 *)

		bAMM_T_Ch_T1HP_MsMs		:= FALSE;		(* A2280 *) (* 2318 *)
		bAMM_T_Ch_T1HP_A_Ms		:= FALSE;		(* W2460 *) (* 2479 *)
		bAMM_T_Ch_T1HP_B_Ms		:= FALSE;		(* W2461 *) (* 2480 *)
		bAMM_T_Ch_T1HP_Lo		:= FALSE;		(* W2531 *) (* 2477 *)

		bAMM_T_Ch_T2HP_Ms		:= FALSE;		(* W2490 *) (* 2491 *)
		bAMM_T_Ch_T2HP_A_Ms		:= FALSE;		(* W2483 *) (* 2485 *)
		bAMM_T_Ch_T2HP_B_Ms		:= FALSE;		(* W2484 *) (* 2486 *)
		bAMM_T_Ch_T2HP_HiHi		:= FALSE;		(* A2368 *)	(* 2369 *)

		bAMM_T_Ch_T2s_MsMs		:= FALSE;		(* A1114 *)
		bAMM_T_Ch_T2s_A_Ms		:= FALSE;		(* W2619 *)
		bAMM_T_Ch_T2s_B_Ms		:= FALSE;		(* W2620 *)
		bAMM_T_Ch_T2s_Lo		:= FALSE;		(* W3562 *)
		bAMM_T_Ch_T2s_A_Lo		:= FALSE;		(* W2510 *)
		bAMM_T_Ch_T2s_B_Lo		:= FALSE;		(* W2512 *)
		bAMM_T_Ch_T2s_Hi		:= FALSE;		(* W3411 *)
		bAMM_T_Ch_T2s_A_Hi		:= FALSE;		(* W2511 *)
		bAMM_T_Ch_T2s_B_Hi		:= FALSE;		(* W2513 *)
		bAMM_T_Ch_T2s_HiHi		:= FALSE;		(* A1040 *)
		bAMM_T_Ch_T2s_A_HiHi	:= FALSE;		(* A2216 *)
		bAMM_T_Ch_T2s_B_HiHi	:= FALSE;		(* A2219 *)
		bAMM_T_Ch_T2s_RocHiHi	:= FALSE;		(* A1105 *)
		bAMM_T_Ch_T2s_A_RocHiHi	:= FALSE;		(* A2217 *)
		bAMM_T_Ch_T2s_B_RocHiHi	:= FALSE;		(* A2220 *)
		bAMM_T_Ch_T2s_DiffHi	:= FALSE;		(* W2525 *)
	END_IF

	rP_Red_Ch_T2s				:= 0;
	rP_Red_Ch_T2s_A				:= 0;
	rP_Red_Ch_T2s_B				:= 0;
	OUT_CH.rP_Red_Ch_T2s_Norm 	:= 1;													(* release full load - no reduction *)
	OUT_CH.rP_Red_Ch_T2HP_Norm 	:= 1;													(* release full load - no reduction *)
	OUT_CH.rP_Red_Ch_T2LP_Norm 	:= 1;													(* release full load - no reduction *)
	OUT_CH.bAMM_T_Ch_T2s_Avg	:= FALSE;												(* collective warning *)
	OUT_CH.bAMM_T_Ch_T1HP_Avg	:= FALSE;												(* collective warning *)
	OUT_CH.bAMM_T_Ch_T1LP_Avg	:= FALSE;												(* collective warning *)
	OUT_CH.bRelEngStart_Ch_T2	:= TRUE;												(* Startfreigabe *)

	(*--------------------------------------------------*)
	(* VISU var of module 								*)
	(*--------------------------------------------------*)
	MM2VIS.rT_Ch_T1LP			:= IN_CH.tT_Ch_T1LP.Ai;
	MM2VIS.rT_Ch_T1LP_A			:= IN_CH.tT_Ch_T1LP_A.Ai;
	MM2VIS.rT_Ch_T1LP_B			:= IN_CH.tT_Ch_T1LP_B.Ai;

	MM2VIS.rT_Ch_T2LP			:= IN_CH.tT_Ch_T2LP.Ai;
	MM2VIS.rT_Ch_T2LP_A			:= IN_CH.tT_Ch_T2LP_A.Ai;
	MM2VIS.rT_Ch_T2LP_B			:= IN_CH.tT_Ch_T2LP_B.Ai;

	MM2VIS.rT_Ch_T1HP			:= IN_CH.tT_Ch_T1HP.Ai;
	MM2VIS.rT_Ch_T1HP_A			:= IN_CH.tT_Ch_T1HP_A.Ai;
	MM2VIS.rT_Ch_T1HP_B			:= IN_CH.tT_Ch_T1HP_B.Ai;

	MM2VIS.rT_Ch_T2HP			:= IN_CH.tT_Ch_T2HP.Ai;
	MM2VIS.rT_Ch_T2HP_A			:= IN_CH.tT_Ch_T2HP_A.Ai;
	MM2VIS.rT_Ch_T2HP_B			:= IN_CH.tT_Ch_T2HP_B.Ai;

	MM2VIS.rT_Ch_T2s			:= IN_CH.tT_Ch_T2s.Ai;
	MM2VIS.rT_Ch_T2s_A			:= IN_CH.tT_Ch_T2s_A.Ai;
	MM2VIS.rT_Ch_T2s_B			:= IN_CH.tT_Ch_T2s_B.Ai;

	(*------------------------------------------------------------------*)
	(* Save actual value every second for RATE OF CHANGE calculation	*)
	(*------------------------------------------------------------------*)
	xTON_1000ms(IN:= NOT xTON_1000ms.Q, PT:= T#980ms);									(* 980ms + 2x cycle time = 1000 ms *)

	IF xTON_1000ms.Q THEN	rT_Ch_T2s_Old	:= IN_CH.tT_Ch_T2s.Ai;
							rT_Ch_T2s_A_Old	:= IN_CH.tT_Ch_T2s_A.Ai;
							rT_Ch_T2s_B_Old	:= IN_CH.tT_Ch_T2s_B.Ai;	END_IF

	(*--------------------------------------------------*)
	(* release for error monitoring 					*)
	(*--------------------------------------------------*)
	IF bRelModul_ParaSetupOk AND IN_CH.tPB2MM.bSys_Run THEN

		(*------------------------------------------------------------------*)
		(* measurement signal failure 										*)
		(*------------------------------------------------------------------*)
		(* charge temperature T1 before low pressure TC *)
		bAMM_T_Ch_T1LP_Ms 	:= Para.bT_Ch_T1LP_Exist   AND NOT IN_CH.tT_Ch_T1LP.GoodQual; 											(* W2411 *)
		bAMM_T_Ch_T1LP_A_Ms	:= Para.bT_Ch_T1LP_A_Exist AND NOT IN_CH.tT_Ch_T1LP_A.GoodQual;											(* W2413 *)
		bAMM_T_Ch_T1LP_B_Ms	:= Para.bT_Ch_T1LP_B_Exist AND NOT IN_CH.tT_Ch_T1LP_B.GoodQual;											(* W2414 *)

			(* release monitoring	*)
			xTON_RelMon_T1LP(IN	 := Para.bT_Ch_T1LP_Exist   AND NOT bAMM_T_Ch_T1LP_Ms, 	 PT:= T#10s);
			xTON_RelMon_T1LP_A(IN:= Para.bT_Ch_T1LP_A_Exist AND NOT bAMM_T_Ch_T1LP_A_Ms, PT:= T#10s);
			xTON_RelMon_T1LP_B(IN:= Para.bT_Ch_T1LP_B_Exist AND NOT bAMM_T_Ch_T1LP_B_Ms, PT:= T#10s);

			bRelMon_T1LP	:= xTON_RelMon_T1LP.Q;				(* delayed reswitch to valid meas.value *)
			bRelMon_T1LP_A	:= xTON_RelMon_T1LP_A.Q;
			bRelMon_T1LP_B	:= xTON_RelMon_T1LP_B.Q;

		(* charge temperature T2 after low pressure TC *)
		bAMM_T_Ch_T2LP_Ms 	:= Para.bT_Ch_T2LP_Exist   AND NOT IN_CH.tT_Ch_T2LP.GoodQual; 											(* W2489 *)
		bAMM_T_Ch_T2LP_A_Ms	:= Para.bT_Ch_T2LP_A_Exist AND NOT IN_CH.tT_Ch_T2LP_A.GoodQual;											(* W2481 *)
		bAMM_T_Ch_T2LP_B_Ms	:= Para.bT_Ch_T2LP_B_Exist AND NOT IN_CH.tT_Ch_T2LP_B.GoodQual;											(* W2482 *)

			(* release monitoring	*)
			xTON_RelMon_T2LP(IN	 := Para.bT_Ch_T2LP_Exist   AND NOT bAMM_T_Ch_T2LP_Ms, 	 PT:= T#10s);
			xTON_RelMon_T2LP_A(IN:= Para.bT_Ch_T2LP_A_Exist AND NOT bAMM_T_Ch_T2LP_A_Ms, PT:= T#10s);
			xTON_RelMon_T2LP_B(IN:= Para.bT_Ch_T2LP_B_Exist AND NOT bAMM_T_Ch_T2LP_B_Ms, PT:= T#10s);

			bRelMon_T2LP	:= xTON_RelMon_T2LP.Q;				(* delayed reswitch to valid meas.value *)
			bRelMon_T2LP_A	:= xTON_RelMon_T2LP_A.Q;
			bRelMon_T2LP_B	:= xTON_RelMon_T2LP_B.Q;

		(* charge temperature T1 before high pressure TC *)
		bAMM_T_Ch_T1HP_A_Ms	:=	  Para.bT_Ch_T1HP_A_Exist AND NOT IN_CH.tT_Ch_T1HP_A.GoodQual;							(* W2460 *)	(* W2479 *)
		bAMM_T_Ch_T1HP_B_Ms	:= 	  Para.bT_Ch_T1HP_B_Exist AND NOT IN_CH.tT_Ch_T1HP_B.GoodQual;							(* W2461 *)	(* W2480 *)
		bAMM_T_Ch_T1HP_MsMs := (  Para.bT_Ch_T1HP_Exist	  AND NOT IN_CH.tT_Ch_T1HP.GoodQual) OR 						(* A2280 *)	(* A2318 *)
							   (((Para.bT_Ch_T1HP_B_Exist AND NOT Para.bT_Ch_T1HP_A_Exist) OR bAMM_T_Ch_T1HP_A_Ms) AND
							    ((Para.bT_Ch_T1HP_A_Exist AND NOT Para.bT_Ch_T1HP_B_Exist) OR bAMM_T_Ch_T1HP_B_Ms)	  );

			(* release monitoring	*)
			xTON_RelMon_T1HP(IN	 := Para.bT_Ch_T1HP_Exist   AND NOT bAMM_T_Ch_T1HP_MsMs, PT:= T#10s);
			xTON_RelMon_T1HP_A(IN:= Para.bT_Ch_T1HP_A_Exist AND NOT bAMM_T_Ch_T1HP_A_Ms, PT:= T#10s);
			xTON_RelMon_T1HP_B(IN:= Para.bT_Ch_T1HP_B_Exist AND NOT bAMM_T_Ch_T1HP_B_Ms, PT:= T#10s);

			bRelMon_T1HP	:= xTON_RelMon_T1HP.Q;				(* delayed reswitch to valid meas.value *)
			bRelMon_T1HP_A	:= xTON_RelMon_T1HP_A.Q;
			bRelMon_T1HP_B	:= xTON_RelMon_T1HP_B.Q;

		(* charge temperature T2 after high pressure TC *)
		bAMM_T_Ch_T2HP_Ms 	:= Para.bT_Ch_T2HP_Exist   AND NOT IN_CH.tT_Ch_T2HP.GoodQual; 								(* W2490 *)	(* W2491 *)
		bAMM_T_Ch_T2HP_A_Ms := Para.bT_Ch_T2HP_A_Exist AND NOT IN_CH.tT_Ch_T2HP_A.GoodQual;								(* W2483 *)	(* W2485 *)
		bAMM_T_Ch_T2HP_B_Ms	:= Para.bT_Ch_T2HP_B_Exist AND NOT IN_CH.tT_Ch_T2HP_B.GoodQual;								(* W2484 *)	(* W2486 *)

			(* release monitoring	*)
			xTON_RelMon_T2HP(IN	 := Para.bT_Ch_T2HP_Exist   AND NOT bAMM_T_Ch_T2HP_Ms,   PT:= T#10s);
			xTON_RelMon_T2HP_A(IN:= Para.bT_Ch_T2HP_A_Exist AND NOT bAMM_T_Ch_T2HP_A_Ms, PT:= T#10s);
			xTON_RelMon_T2HP_B(IN:= Para.bT_Ch_T2HP_B_Exist AND NOT bAMM_T_Ch_T2HP_B_Ms, PT:= T#10s);

			bRelMon_T2HP	:= xTON_RelMon_T2HP.Q;				(* delayed reswitch to valid meas.value *)
			bRelMon_T2HP_A	:= xTON_RelMon_T2HP_A.Q;
			bRelMon_T2HP_B	:= xTON_RelMon_T2HP_B.Q;

		(* charge temperature T2' *)
		bAMM_T_Ch_T2s_A_Ms 	:= 	  Para.bT_Ch_T2s_A_Exist AND NOT IN_CH.tT_Ch_T2s_A.GoodQual;										(* W2619 *)
		bAMM_T_Ch_T2s_B_Ms 	:= 	  Para.bT_Ch_T2s_B_Exist AND NOT IN_CH.tT_Ch_T2s_B.GoodQual;										(* W2620 *)
		bAMM_T_Ch_T2s_MsMs 	:= (  Para.bT_Ch_T2s_Exist   AND NOT IN_CH.tT_Ch_T2s.GoodQual) 	OR										(* A1114 *)
							   (((Para.bT_Ch_T2s_B_Exist AND NOT Para.bT_Ch_T2s_A_Exist) OR bAMM_T_Ch_T2s_A_Ms) AND
							    ((Para.bT_Ch_T2s_A_Exist AND NOT Para.bT_Ch_T2s_B_Exist) OR bAMM_T_Ch_T2s_B_Ms)	  );

			(* release monitoring	*)
			xTON_RelMon_T2s(IN	:= Para.bT_Ch_T2s_Exist   AND NOT bAMM_T_Ch_T2s_MsMs, PT:= T#10s);
			xTON_RelMon_T2s_A(IN:= Para.bT_Ch_T2s_A_Exist AND NOT bAMM_T_Ch_T2s_A_Ms, PT:= T#10s);
			xTON_RelMon_T2s_B(IN:= Para.bT_Ch_T2s_B_Exist AND NOT bAMM_T_Ch_T2s_B_Ms, PT:= T#10s);

			bRelMon_T2s		:= xTON_RelMon_T2s.Q;				(* delayed reswitch to valid meas.value *)
			bRelMon_T2s_A	:= xTON_RelMon_T2s_A.Q;
			bRelMon_T2s_B	:= xTON_RelMon_T2s_B.Q;

		(*------------------------------------------------------------------*)
		(* temperature MIN		 											*)
		(*------------------------------------------------------------------*)
	  	(* charge temperature T1 before high pressure TC minimum *)
		IF bP_Nom10_300s THEN
			bAMM_T_Ch_T1HP_Lo	:= ((IN_CH.tT_Ch_T1HP.Ai   < Para.rT_Ch_T1HP_Lo) AND bRelMon_T1HP  ) OR					(* W2531 *)	(* W2477 *)
								   ((IN_CH.tT_Ch_T1HP_A.Ai < Para.rT_Ch_T1HP_Lo) AND bRelMon_T1HP_A) OR
						   		   ((IN_CH.tT_Ch_T1HP_B.Ai < Para.rT_Ch_T1HP_Lo) AND bRelMon_T1HP_B);
		END_IF

		(* charge temperature T2' minimum *)
		IF bP_Nom10_600s THEN
			bAMM_T_Ch_T2s_Lo 	:= (IN_CH.tT_Ch_T2s.Ai 	 < Para.rT_Ch_T2s_Lo) AND bRelMon_T2s;										(* W3562 *)
			bAMM_T_Ch_T2s_A_Lo 	:= (IN_CH.tT_Ch_T2s_A.Ai < Para.rT_Ch_T2s_Lo) AND bRelMon_T2s_A;									(* W2510 *)
			bAMM_T_Ch_T2s_B_Lo 	:= (IN_CH.tT_Ch_T2s_B.Ai < Para.rT_Ch_T2s_Lo) AND bRelMon_T2s_B;									(* W2512 *)
	  	END_IF

		(*------------------------------------------------------------------*)
		(* temperature MAX	 / POWER REDUCTION								*)
		(*------------------------------------------------------------------*)
		(* charge temperature T1 before low-pressure TC (air intake) - maximum *)
		IF bRelMon_T1LP OR bRelMon_T1LP_A
						OR bRelMon_T1LP_B  		THEN rT_Ch_T1LP_Max			:= MAX(IN_CH.tT_Ch_T1LP.Ai   * BOOL_TO_REAL(bRelMon_T1LP),
																			 	   IN_CH.tT_Ch_T1LP_A.Ai * BOOL_TO_REAL(bRelMon_T1LP_A),
																			   	   IN_CH.tT_Ch_T1LP_B.Ai * BOOL_TO_REAL(bRelMon_T1LP_B));
												ELSE rT_Ch_T1LP_Max			:= 0;
													 bAMM_T_Ch_T2_Calc		:= Para.bTSTC_Exist AND		(* Engine start blocked *)	(* W9370 *)
																			   Para.bCh_T2Calc_Active;
		END_IF

		(* charge temperature T2 after low-pressure TC - maximum *)
		IF Para.bCh_T2Calc_Active 	AND NOT bRelMon_T2LP
									AND NOT bRelMon_T2LP_A
									AND NOT bRelMon_T2LP_B
									AND 	Para.bTSTC_Exist
		THEN
			(* Find most suitable pressure close to TC *)
			IF	  NOT OUT_CH.bAMM_Pr_Ch_P2LP_Avg	THEN rPr_aLPTC			:= OUT_CH.rPr_Ch_P2LP_Max;
			ELSIF NOT OUT_CH.bAMM_Pr_Ch_P1HP_Avg	THEN rPr_aLPTC			:= OUT_CH.rPr_Ch_P1HP_Max + Para.rDPr_Ch_T2Calc_LP_Cooler;
													ELSE rPr_aLPTC			:= 0;
														 bAMM_T_Ch_T2_Calc	:= TRUE;					(* Engine start blocked *)	(* W9370 *)
			END_IF

			IF	  NOT OUT_CH.bAMM_Pr_Ch_P1LP_Avg	THEN rPr_bLPTC			:= OUT_CH.rPr_Ch_P1LP_Max;
			ELSIF NOT IN_CH.bAMM_Pr_Baro_Internal	THEN rPr_bLPTC			:= IN_CH.rPr_Baro_Internal  - Para.rDPr_Ch_T2Calc_AirFilt;
			ELSIF NOT bAMM_T_Ch_T2_Calc 	AND
					  IN_CH.rN_EngAct < 10			THEN rPr_bLPTC			:= rPr_aLPTC 				- Para.rDPr_Ch_T2Calc_AirFilt;
			END_IF

			(* calculation - T2 after low-pressure TC *)
			IF 	NOT bAMM_T_Ch_T2_Calc 			AND														(* Engine start released *)
				Para.rPc_Ch_T2Calc_LP_Eff <> 0	AND														(* no division by zero *)
				rPr_bLPTC 				  <> 0		THEN rT_Ch_T2LP_Max		:= (rT_Ch_T1LP_Max + 273.15) / Para.rPc_Ch_T2Calc_LP_Eff *
								  											   ((rPr_aLPTC / rPr_bLPTC)**(0.38 / 1.38) - 1) + rT_Ch_T1LP_Max;
													ELSE rT_Ch_T2LP_Max		:= 0;
														 bAMM_T_Ch_T2_Calc	:= TRUE;					(* Engine start blocked *)	(* W9370 *)
			END_IF

			MM2VIS.rT_Ch_T2LP_Calc	:= rT_Ch_T2LP_Max * BOOL_TO_REAL(bStartSpd);						(* calculation only used during operation *)
		ELSE
			MM2VIS.rT_Ch_T2LP_Calc	:= 0;
			rT_Ch_T2LP_Max			:= MAX(IN_CH.tT_Ch_T2LP.Ai   * BOOL_TO_REAL(bRelMon_T2LP),
										   IN_CH.tT_Ch_T2LP_A.Ai * BOOL_TO_REAL(bRelMon_T2LP_A),
										   IN_CH.tT_Ch_T2LP_B.Ai * BOOL_TO_REAL(bRelMon_T2LP_B));
		END_IF

			(* power reduction of 4% per °C deviation to at least 80% *)
			xSigScal_R_P_Red_Ch_T2LP.X	:= rT_Ch_T2LP_Max;
			xSigScal_R_P_Red_Ch_T2LP.X1 := Para.rT_Ch_T2LP_HiHi - 5;
			xSigScal_R_P_Red_Ch_T2LP.X2	:= Para.rT_Ch_T2LP_HiHi;
			xSigScal_R_P_Red_Ch_T2LP.Y1 := 1.0;
			xSigScal_R_P_Red_Ch_T2LP.Y2 := 0.8;
			xSigScal_R_P_Red_Ch_T2LP();

			xRAMPE_R_P_Red_Ch_T2LP(In	:= xSigScal_R_P_Red_Ch_T2LP.Y_SCAL, enable := bStartSpd);

		IF Para.bCh_T2Calc_Active AND Para.bTSTC_Exist THEN
			OUT_CH.rP_Red_Ch_T2LP_Norm	:= LIMIT(0.8, xRAMPE_R_P_Red_Ch_T2LP.Out, 1);												(* B9075 *)
		END_IF

		bAMM_T_Ch_T2LP_HiHi				:= rT_Ch_T2LP_Max > Para.rT_Ch_T2LP_HiHi AND Para.bTSTC_Exist;								(* A2370 *)

		(* charge temperature T1 before high pressure TC maximum *)
		IF bRelMon_T1HP OR bRelMon_T1HP_A
						OR bRelMon_T1HP_B		THEN rT_Ch_T1HP_Max			:= MAX(IN_CH.tT_Ch_T1HP.Ai   * BOOL_TO_REAL(bRelMon_T1HP),
									   											   IN_CH.tT_Ch_T1HP_A.Ai * BOOL_TO_REAL(bRelMon_T1HP_A),
																				   IN_CH.tT_Ch_T1HP_B.Ai * BOOL_TO_REAL(bRelMon_T1HP_B));
		ELSIF 	NOT Para.bTSTC_Exist 		AND
				NOT Para.bT_Ch_T1HP_Exist 	AND
				NOT Para.bT_Ch_T1HP_A_Exist AND
				NOT Para.bT_Ch_T1HP_B_Exist	AND
					(bRelMon_T1LP 	OR
				 	 bRelMon_T1LP_A OR
					 bRelMon_T1LP_B	  ) 		THEN rT_Ch_T1HP_Max			:= rT_Ch_T1LP_Max;			(* Use intake air temperature if T1HP is not available *)
												ELSE rT_Ch_T1HP_Max			:= 0;
													 bAMM_T_Ch_T2_Calc		:= Para.bCh_T2Calc_Active;	(* Engine start blocked *)	(* W9370 *)
		END_IF

		(* charge temperature T2 after high-pressure TC - maximum *)
		IF Para.bCh_T2Calc_Active 	AND NOT bRelMon_T2HP
									AND NOT bRelMon_T2HP_A
									AND NOT bRelMon_T2HP_B
		THEN
			(* Find most suitable pressure close to TC *)
			IF	  NOT OUT_CH.bAMM_Pr_Ch_P2HP_Avg	THEN rPr_aHPTC			:= OUT_CH.rPr_Ch_P2HP_Max;
			ELSIF NOT OUT_CH.bAMM_Pr_Ch_P2_Avg		THEN rPr_aHPTC			:= OUT_CH.rPr_Ch_P2_Max  + Para.rDPr_Ch_T2Calc_HP_Cooler;
			ELSIF NOT OUT_CH.bAMM_Pr_Ch_P2s_Avg		THEN rPr_aHPTC			:= OUT_CH.rPr_Ch_P2s_Max + Para.rDPr_Ch_T2Calc_HP_Cooler;
													ELSE rPr_aHPTC			:= 0;
														 bAMM_T_Ch_T2_Calc	:= TRUE;					(* Engine start blocked *)	(* W9370 *)
				END_IF

			IF Para.bTSTC_Exist THEN
				IF	  NOT OUT_CH.bAMM_Pr_Ch_P1HP_Avg	THEN rPr_bHPTC		:= OUT_CH.rPr_Ch_P1HP_Max;
				ELSIF NOT OUT_CH.bAMM_Pr_Ch_P2LP_Avg	THEN rPr_bHPTC		:= OUT_CH.rPr_Ch_P2LP_Max - Para.rDPr_Ch_T2Calc_LP_Cooler;
														ELSE rPr_bHPTC		:= 0;
													 	 bAMM_T_Ch_T2_Calc	:= TRUE;					(* Engine start blocked *)	(* W9370 *)
				END_IF
			ELSE
				IF	  NOT OUT_CH.bAMM_Pr_Ch_P1HP_Avg	THEN rPr_bHPTC		:= OUT_CH.rPr_Ch_P1HP_Max;
				ELSIF NOT OUT_CH.bAMM_Pr_Ch_P1LP_Avg	THEN rPr_bHPTC		:= OUT_CH.rPr_Ch_P1LP_Max;
				ELSIF NOT IN_CH.bAMM_Pr_Baro_Internal	THEN rPr_bHPTC		:= IN_CH.rPr_Baro_Internal	- Para.rDPr_Ch_T2Calc_AirFilt;
				ELSIF NOT bAMM_T_Ch_T2_Calc 	AND
						  IN_CH.rN_EngAct < 10			THEN rPr_bHPTC		:= rPr_aHPTC 				- Para.rDPr_Ch_T2Calc_AirFilt;
				END_IF
			END_IF

			(* calculation - T2 after high-pressure TC *)
			IF 	NOT bAMM_T_Ch_T2_Calc 			AND														(* Engine start released *)
				Para.rPc_Ch_T2Calc_HP_Eff <> 0	AND														(* no division by zero *)
				rPr_bHPTC 				  <> 0		THEN rT_Ch_T2HP_Max		:= (rT_Ch_T1HP_Max + 273.15) / Para.rPc_Ch_T2Calc_HP_Eff *
																			   ((rPr_aHPTC / rPr_bHPTC)**(0.38 / 1.38) - 1) + rT_Ch_T1HP_Max;
													ELSE rT_Ch_T2HP_Max		:= 0;
														 bAMM_T_Ch_T2_Calc	:= TRUE;					(* Engine start blocked *)	(* W9370 *)
			END_IF

			MM2VIS.rT_Ch_T2HP_Calc	:= rT_Ch_T2HP_Max * BOOL_TO_REAL(bStartSpd);						(* calculation only used during operation *)
		ELSE
			MM2VIS.rT_Ch_T2HP_Calc	:= 0;
			rT_Ch_T2HP_Max			:= MAX(IN_CH.tT_Ch_T2HP.Ai   * BOOL_TO_REAL(bRelMon_T2HP),
										   IN_CH.tT_Ch_T2HP_A.Ai * BOOL_TO_REAL(bRelMon_T2HP_A),
										   IN_CH.tT_Ch_T2HP_B.Ai * BOOL_TO_REAL(bRelMon_T2HP_B));
		END_IF

			(* power reduction of 4% per °C deviation to at least 80% *)
			xSigScal_R_P_Red_Ch_T2HP.X	:= rT_Ch_T2HP_Max;
			xSigScal_R_P_Red_Ch_T2HP.X1 := Para.rT_Ch_T2HP_HiHi - 5;
			xSigScal_R_P_Red_Ch_T2HP.X2	:= Para.rT_Ch_T2HP_HiHi;
			xSigScal_R_P_Red_Ch_T2HP.Y1 := 1.0;
			xSigScal_R_P_Red_Ch_T2HP.Y2 := 0.8;
			xSigScal_R_P_Red_Ch_T2HP();

			xRAMPE_R_P_Red_Ch_T2HP(In	:= xSigScal_R_P_Red_Ch_T2HP.Y_SCAL, enable := bStartSpd);

		IF Para.bCh_T2Calc_Active THEN
			OUT_CH.rP_Red_Ch_T2HP_Norm	:= LIMIT(0.8, xRAMPE_R_P_Red_Ch_T2HP.Out, 1);											(* B9075 *)
		END_IF

		bAMM_T_Ch_T2HP_HiHi				:= rT_Ch_T2HP_Max > Para.rT_Ch_T2HP_HiHi;										(* A2368 *)	(* A2369 *)
		OUT_CH.bRelEngStart_Ch_T2		:= NOT bAMM_T_Ch_T2_Calc;										(* Engine start released *)

		(* interpolation of T2' temperature max parameter *)
		Para.rT_Ch_T2s_Hi[0] 	:= Para.rT_Ch_T2s_Hi[1]  + (IN_CH.rGT_QualMix_1_2 * (Para.rT_Ch_T2s_Hi[2]  - Para.rT_Ch_T2s_Hi[1] ));
		Para.rP_Red_Ch_T2s[0]	:= Para.rP_Red_Ch_T2s[1] + (IN_CH.rGT_QualMix_1_2 * (Para.rP_Red_Ch_T2s[2] - Para.rP_Red_Ch_T2s[1]));

		Para.rT_Ch_T2s_Hi[0]	:= Para.rT_Ch_T2s_Hi[0]  + (IN_CH.rGT_RatioMix 	  * (Para.rT_Ch_T2s_Hi[3]  - Para.rT_Ch_T2s_Hi[0] ));
		Para.rP_Red_Ch_T2s[0] 	:= Para.rP_Red_Ch_T2s[0] + (IN_CH.rGT_RatioMix 	  * (Para.rP_Red_Ch_T2s[3] - Para.rP_Red_Ch_T2s[0]));

		(* charge temperature T2' maximum -> start power reduction *)
		IF bNetP_Island_20s
		THEN
			bAMM_T_Ch_T2s_Hi 	:= (IN_CH.tT_Ch_T2s.Ai 	 > Para.rT_Ch_T2s_Hi[gastype]) AND bRelMon_T2s; 							(* W3411 *)
			bAMM_T_Ch_T2s_A_Hi	:= (IN_CH.tT_Ch_T2s_A.Ai > Para.rT_Ch_T2s_Hi[gastype]) AND bRelMon_T2s_A;							(* W2511 *)
			bAMM_T_Ch_T2s_B_Hi	:= (IN_CH.tT_Ch_T2s_B.Ai > Para.rT_Ch_T2s_Hi[gastype]) AND bRelMon_T2s_B;							(* W2513 *)
		END_IF

			(* Power reduction per °C inclination *) 																				(* B2126 *)
			IF bAMM_T_Ch_T2s_Hi OR bAMM_T_Ch_T2s_A_Hi OR bAMM_T_Ch_T2s_B_Hi
			THEN
				IF bAMM_T_Ch_T2s_Hi	  THEN rP_Red_Ch_T2s   := (IN_CH.tT_Ch_T2s.Ai   - Para.rT_Ch_T2s_Hi[gastype]) *
																				 	  Para.rP_Red_Ch_T2s[gastype]; 	END_IF
				IF bAMM_T_Ch_T2s_A_Hi THEN rP_Red_Ch_T2s_A := (IN_CH.tT_Ch_T2s_A.Ai - Para.rT_Ch_T2s_Hi[gastype]) *
																				  	  Para.rP_Red_Ch_T2s[gastype]; 	END_IF
				IF bAMM_T_Ch_T2s_B_Hi THEN rP_Red_Ch_T2s_B := (IN_CH.tT_Ch_T2s_B.Ai - Para.rT_Ch_T2s_Hi[gastype]) *
																				  	  Para.rP_Red_Ch_T2s[gastype]; 	END_IF
				(* power reduction initiating at actual power *)
				OUT_CH.rP_Red_Ch_T2s_Norm := LIMIT(0, rP_Act_Norm_SaveT2s - MAX(rP_Red_Ch_T2s, rP_Red_Ch_T2s_A, rP_Red_Ch_T2s_B), 1);
			ELSE
				rP_Act_Norm_SaveT2s		  := IN_CH.rP_Act_Norm_Filt_TC2;				(* save actual power *)
			END_IF

		(* charge temperature T2' maximum -> ERROR *)
		IF bNetP_Island_20s
		THEN
			bAMM_T_Ch_T2s_HiHi 		:= (IN_CH.tT_Ch_T2s.Ai 	 > Para.rT_Ch_T2s_HiHi) AND bRelMon_T2s;								(* A1040 *)
			bAMM_T_Ch_T2s_A_HiHi	:= (IN_CH.tT_Ch_T2s_A.Ai > Para.rT_Ch_T2s_HiHi) AND bRelMon_T2s_A;								(* A2216 *)
			bAMM_T_Ch_T2s_B_HiHi 	:= (IN_CH.tT_Ch_T2s_B.Ai > Para.rT_Ch_T2s_HiHi) AND bRelMon_T2s_B;								(* A2219 *)
		END_IF

		(*------------------------------------------------------------------*)
		(* temperature RATE OF CHANGE maximum (Änderungsgeschwindigkeit)	*)
		(*------------------------------------------------------------------*)
			(* Release monitoring	*)
			IF IN_CH.tEng_Run.Do 	THEN bRelMon_T2s_Roc := TRUE; 	END_IF
			IF NOT bStartSpd 		THEN bRelMon_T2s_Roc := FALSE; 	END_IF

		(* charge temperature T2' *)
		IF bRelMon_T2s_Roc THEN
			bAMM_T_Ch_T2s_RocHiHi	:= ((IN_CH.tT_Ch_T2s.Ai   - rT_Ch_T2s_Old) 	 > Para.rT_Ch_T2s_Roc_HiHi) AND bRelMon_T2s;		(* A1105 *)
			bAMM_T_Ch_T2s_A_RocHiHi	:= ((IN_CH.tT_Ch_T2s_A.Ai - rT_Ch_T2s_A_Old) > Para.rT_Ch_T2s_Roc_HiHi) AND bRelMon_T2s_A;		(* A2217 *)
			bAMM_T_Ch_T2s_B_RocHiHi	:= ((IN_CH.tT_Ch_T2s_B.Ai - rT_Ch_T2s_B_Old) > Para.rT_Ch_T2s_Roc_HiHi) AND bRelMon_T2s_B;		(* A2220 *)
		END_IF

		(*------------------------------------------------------------------*)
		(* temperature INCLINATION maximum (Spreizung)						*)
		(*------------------------------------------------------------------*)
		(* charge temperature T2' *)
		IF bP_Nom10_60s THEN
			bAMM_T_Ch_T2s_DiffHi 	:= (ABS(IN_CH.tT_Ch_T2s_A.Ai - IN_CH.tT_Ch_T2s_B.Ai) > Para.rT_Ch_T2s_Diff_Hi)	AND				(* W2525 *)
								   		bRelMon_T2s_A AND bRelMon_T2s_B;
		END_IF

		(*----------------------------------------------------------------------------------------------------------------------------------*)
		(* Handover charge temperature to other modules																						*)
		(*----------------------------------------------------------------------------------------------------------------------------------*)
		(* charge temperature before low-pressure TC *)
		IF 		bRelMon_T1LP	THEN  OUT_CH.rT_Ch_T1LP_Avg		:= IN_CH.tT_Ch_T1LP.Ai;
		ELSIF 	bRelMon_T1LP_A	THEN
			IF 	bRelMon_T1LP_B	THEN  OUT_CH.rT_Ch_T1LP_Avg		:=(IN_CH.tT_Ch_T1LP_A.Ai + IN_CH.tT_Ch_T1LP_B.Ai) / 2;
								ELSE  OUT_CH.rT_Ch_T1LP_Avg 	:= IN_CH.tT_Ch_T1LP_A.Ai;
			END_IF
		ELSIF 	bRelMon_T1LP_B	THEN  OUT_CH.rT_Ch_T1LP_Avg 	:= IN_CH.tT_Ch_T1LP_B.Ai;
								ELSE  OUT_CH.rT_Ch_T1LP_Avg 	:= 0;
									  OUT_CH.bAMM_T_Ch_T1LP_Avg	:= TRUE;
		END_IF

		MM2VIS.rT_Ch_T1LP_Avg	:= OUT_CH.rT_Ch_T1LP_Avg;				(* VISU *)

		(* charge temperature before high-pressure TC *)
		IF 		bRelMon_T1HP	THEN  OUT_CH.rT_Ch_T1HP_Avg		:= IN_CH.tT_Ch_T1HP.Ai;
		ELSIF 	bRelMon_T1HP_A	THEN
			IF 	bRelMon_T1HP_B	THEN  OUT_CH.rT_Ch_T1HP_Avg		:=(IN_CH.tT_Ch_T1HP_A.Ai + IN_CH.tT_Ch_T1HP_B.Ai) / 2;
								ELSE  OUT_CH.rT_Ch_T1HP_Avg 	:= IN_CH.tT_Ch_T1HP_A.Ai;
			END_IF
		ELSIF 	bRelMon_T1HP_B	THEN  OUT_CH.rT_Ch_T1HP_Avg 	:= IN_CH.tT_Ch_T1HP_B.Ai;
								ELSE  OUT_CH.rT_Ch_T1HP_Avg 	:= 0;
									  OUT_CH.bAMM_T_Ch_T1HP_Avg	:= TRUE;
		END_IF

		MM2VIS.rT_Ch_T1HP_Avg	:= OUT_CH.rT_Ch_T1HP_Avg;				(* VISU *)

		(* charge temperature t2' *)
		IF 	 bRelMon_T2s		THEN	OUT_CH.rT_Ch_T2s_Avg_UF	:= IN_CH.tT_Ch_T2s.Unfilt;
										OUT_CH.rT_Ch_T2s_Avg 	:= IN_CH.tT_Ch_T2s.Ai;
										OUT_CH.rT_Ch_T2s_A 		:= 0;
										OUT_CH.rT_Ch_T2s_B 		:= 0;
		ELSIF  	 bRelMon_T2s_A	THEN
			IF 	 bRelMon_T2s_B 	THEN 	OUT_CH.rT_Ch_T2s_Avg_UF	:=(IN_CH.tT_Ch_T2s_A.Unfilt + IN_CH.tT_Ch_T2s_B.Unfilt) / 2;
										OUT_CH.rT_Ch_T2s_Avg	:=(IN_CH.tT_Ch_T2s_A.Ai     + IN_CH.tT_Ch_T2s_B.Ai) 	/ 2;
										OUT_CH.rT_Ch_T2s_A 		:= IN_CH.tT_Ch_T2s_A.Ai;
										OUT_CH.rT_Ch_T2s_B 		:= IN_CH.tT_Ch_T2s_B.Ai;

								ELSE	OUT_CH.rT_Ch_T2s_Avg_UF	:= IN_CH.tT_Ch_T2s_A.Unfilt;
										OUT_CH.rT_Ch_T2s_Avg 	:= IN_CH.tT_Ch_T2s_A.Ai;
										OUT_CH.rT_Ch_T2s_A 		:= IN_CH.tT_Ch_T2s_A.Ai;
										OUT_CH.rT_Ch_T2s_B 		:= IN_CH.tT_Ch_T2s_A.Ai;
			END_IF

		ELSIF  	bRelMon_T2s_B 	THEN 	OUT_CH.rT_Ch_T2s_Avg_UF := IN_CH.tT_Ch_T2s_B.Unfilt;
										OUT_CH.rT_Ch_T2s_Avg 	:= IN_CH.tT_Ch_T2s_B.Ai;
										OUT_CH.rT_Ch_T2s_A 		:= IN_CH.tT_Ch_T2s_B.Ai;
										OUT_CH.rT_Ch_T2s_B 		:= IN_CH.tT_Ch_T2s_B.Ai;

								 ELSE	(* J920: Handover parameter-value if both sensors with error *)
										OUT_CH.rT_Ch_T2s_Avg_UF	:= Para.rT_Ch_T2s_Hi[gastype] * BOOL_TO_REAL(xEngType.Type9);
										OUT_CH.rT_Ch_T2s_Avg 	:= Para.rT_Ch_T2s_Hi[gastype] * BOOL_TO_REAL(xEngType.Type9);
										OUT_CH.rT_Ch_T2s_A 		:= Para.rT_Ch_T2s_Hi[gastype] * BOOL_TO_REAL(xEngType.Type9);
										OUT_CH.rT_Ch_T2s_B 		:= Para.rT_Ch_T2s_Hi[gastype] * BOOL_TO_REAL(xEngType.Type9);
										OUT_CH.bAMM_T_Ch_T2s_Avg:= NOT xEngType.Type9;
		END_IF

		MM2VIS.rT_Ch_T2s_Avg := OUT_CH.rT_Ch_T2s_Avg;					(* VISU *)

	ELSE
		xTON_RelMon_T1LP(IN	 := FALSE);
		xTON_RelMon_T1LP_A(IN:= FALSE);
		xTON_RelMon_T1LP_B(IN:= FALSE);
		xTON_RelMon_T2LP(IN	 := FALSE);
		xTON_RelMon_T2LP_A(IN:= FALSE);
		xTON_RelMon_T2LP_B(IN:= FALSE);
		xTON_RelMon_T1HP(IN	 := FALSE);
		xTON_RelMon_T1HP_A(IN:= FALSE);
		xTON_RelMon_T1HP_B(IN:= FALSE);
		xTON_RelMon_T2HP(IN	 := FALSE);
		xTON_RelMon_T2HP_A(IN:= FALSE);
		xTON_RelMon_T2HP_B(IN:= FALSE);
		xTON_RelMon_T2s(IN	 := FALSE);
		xTON_RelMon_T2s_A(IN := FALSE);
		xTON_RelMon_T2s_B(IN := FALSE);
	END_IF

END_PROGRAM
```

#### CH_Temp.var - Local variables
```iecst
VAR
	bRelMon_T1HP : BOOL := FALSE; (*Release monitoring charge temperature before HP TC *)
	bRelMon_T1HP_A : BOOL := FALSE; (*Release monitoring charge temperature before HP TC A*)
	bRelMon_T1HP_B : BOOL := FALSE; (*Release monitoring charge temperature before HP TC  B*)
	bRelMon_T1LP : BOOL := FALSE; (*Release monitoring charge temperature before LP TC (air intake)*)
	bRelMon_T1LP_A : BOOL := FALSE; (*Release monitoring charge temperature before LP TC A (air intake)*)
	bRelMon_T1LP_B : BOOL := FALSE; (*Release monitoring charge temperature before LP TC  B (air intake)*)
	bRelMon_T2HP : BOOL := FALSE; (*Release monitoring charge temperature after HP TC *)
	bRelMon_T2HP_A : BOOL := FALSE; (*Release monitoring charge temperature after HP TC A*)
	bRelMon_T2HP_B : BOOL := FALSE; (*Release monitoring charge temperature after HP TC  B*)
	bRelMon_T2LP : BOOL := FALSE; (*Release monitoring charge temperature after LP TC*)
	bRelMon_T2LP_A : BOOL := FALSE; (*Release monitoring charge temperature after LP TC A*)
	bRelMon_T2LP_B : BOOL := FALSE; (*Release monitoring charge temperature after LP TC  B*)
	bRelMon_T2s : BOOL := FALSE; (*Release monitoring charge temperature t2' *)
	bRelMon_T2s_A : BOOL := FALSE; (*Release monitoring charge temperature t2' A*)
	bRelMon_T2s_B : BOOL := FALSE; (*Release monitoring charge temperature t2' B*)
	bRelMon_T2s_Roc : BOOL := FALSE; (*Release "rate of change" monitoring for charge temperature t2' *)
	rPr_aHPTC : REAL := 0.0; (*Pressure after high-pressure TC - for calculation*)
	rPr_aLPTC : REAL := 0.0; (*Pressure after low-pressure TC - for calculation*)
	rPr_bHPTC : REAL := 0.0; (*Pressure before high-pressure TC - for calculation*)
	rPr_bLPTC : REAL := 0.0; (*Pressure before low-pressure TC - for calculation*)
	rP_Act_Norm_SaveT2s : REAL := 0.0; (*Save actual power for power reduction by temperature t2' [%Pnom]*)
	rP_Red_Ch_T2s : REAL := 0.0; (*value for power reduction by charge temperature t2' [%Pnom]*)
	rP_Red_Ch_T2s_A : REAL := 0.0; (*value for power reduction by charge temperature t2'  A [%Pnom]*)
	rP_Red_Ch_T2s_B : REAL := 0.0; (*value for power reduction by charge temperature t2'  B [%Pnom]*)
	rT_Ch_T2HP_Max : REAL; (*maximum value - charge temperature after high-pressure TC *) (*V04.12.00.00*)
	rT_Ch_T2LP_Max : REAL; (*maximum value - charge temperature after low-pressure TC *) (*V04.12.00.00*)
	rT_Ch_T2s_A_Old : REAL := 0.0; (*Save charge temperature t2' A for 1 second [°C]*)
	rT_Ch_T2s_B_Old : REAL := 0.0; (*Save charge temperature t2' B for 1 second [°C]*)
	rT_Ch_T2s_Old : REAL := 0.0; (*Save charge temperature t2' for 1 second [°C]*)
END_VAR
VAR CONSTANT
	TASK_TIME_10MS : UINT := 10; (*Taskklassen Zeit 10ms *)
END_VAR
VAR
	xRAMPE_R_P_Red_Ch_T2HP : RAMPE_R := (0); (*FuB*)
	xRAMPE_R_P_Red_Ch_T2LP : RAMPE_R := (0); (*FuB*)
	xSigScal_R_P_Red_Ch_T2HP : xSigScal_R := (0); (*FuB*)
	xSigScal_R_P_Red_Ch_T2LP : xSigScal_R := (0); (*FuB*)
	xTON_200msTick : TON := (0); (*FuB*)
	xTON_1000ms : TON := (0); (*FuB*)
	xTON_RelMon_T1HP : TON := (0); (*FuB*)
	xTON_RelMon_T1HP_A : TON := (0); (*FuB*)
	xTON_RelMon_T1HP_B : TON := (0); (*FuB*)
	xTON_RelMon_T1LP : TON := (0); (*FuB*)
	xTON_RelMon_T1LP_A : TON := (0); (*FuB*)
	xTON_RelMon_T1LP_B : TON := (0); (*FuB*)
	xTON_RelMon_T2HP : TON := (0); (*FuB*)
	xTON_RelMon_T2HP_A : TON := (0); (*FuB*)
	xTON_RelMon_T2HP_B : TON := (0); (*FuB*)
	xTON_RelMon_T2LP : TON := (0); (*FuB*)
	xTON_RelMon_T2LP_A : TON := (0); (*FuB*)
	xTON_RelMon_T2LP_B : TON := (0); (*FuB*)
	xTON_RelMon_T2s : TON := (0); (*FuB*)
	xTON_RelMon_T2s_A : TON := (0); (*FuB*)
	xTON_RelMon_T2s_B : TON := (0); (*FuB*)
END_VAR
```

### Program Logical/ChargingUnit/CH_Press (IEC, version 4.14.0) - charging pressure

#### CH_PressCyclic.st - Cyclic code
```iecst
(*************************************************************************************************************************************
CH_Press	 		 Charging pressures

This code is confidential and proprietary to the INNIO Company.
It may not be used in any form, or reproduced in any manner,
without written permission of the INNIO Company.
Copyright, INNIO Company, 2021

Customized modifications: -
------------------------

History:
-------
V03.99.00.00	19.09.2012	Tinello		restructured
V04.04.00.00	31.10.2016	Tinello		add Pr_Ch_P1LP,Pr_Ch_P2LP, Pr_Ch_P2HP, Pr_Ch_P2bFA -> Spec. (b) & (c)
V04.05.00.00	12.07.2017	Tinello		SWAT 3/J920 -> Spec (d)
V04.05.02.00	16.04.2018	Tinello		enable P2s value forwarding to other SW modules also in op.switch OFF mode
V04.07.00.00	24.03.2019	Tinello		MsErr active with op.switch OFF mode / Calculation of difference pressure adjusted
										Pressure average values forwarding to other SW modules -> Spec (e)
V04.10.00.00	27.01.2021	Tinello		BugFix: Timer-FuB's
V04.12.00.00	25.01.2023	Tinello		Pressure maximum values forwarding to other SW modules
V04.14.00.00    20.06.2024	Soto		Pressure signals plausibility check during standstill

(************************************************************************************************************************************)
PROGRAM _INIT
	rPr_Ch_Max 		:= 1.3;
	rPr_Ch_Min 		:= 0.8;
	rPr_Ch_devMax 	:= 0.08;
	iPr_Ch_lgt 		:= 18;
	tPr_Ch[0].Tag 	:= 'E.08-PI-001';
	tPr_Ch[1].Tag 	:= 'M.05-PI-150';
	tPr_Ch[2].Tag 	:= 'M.05-PI-250';
	tPr_Ch[3].Tag 	:= 'E.08-PI-002';
	tPr_Ch[4].Tag 	:= 'M.05-PI-151';
	tPr_Ch[5].Tag 	:= 'M.05-PI-251';
	tPr_Ch[6].Tag 	:= 'M.08-PI-011';
	tPr_Ch[7].Tag 	:= 'M.05-PI-147';
	tPr_Ch[8].Tag 	:= 'M.05-PI-247';
	tPr_Ch[9].Tag 	:= 'E.08-PI-003';
	tPr_Ch[10].Tag 	:= 'E.08-PI-004';
	tPr_Ch[11].Tag 	:= 'M.05-PI-149';
	tPr_Ch[12].Tag 	:= 'M.05-PI-249';
	tPr_Ch[13].Tag 	:= 'M.08-PI-007';
	tPr_Ch[14].Tag 	:= 'M.08-PI-007/M.05-PI-148';
	tPr_Ch[15].Tag 	:= 'M.08-PI-008/M.05-PI-248';
	tPr_Ch[16].Tag 	:= 'M.05-PI-146';
	tPr_Ch[17].Tag 	:= 'M.05-PI-246';
END_PROGRAM

PROGRAM _CYCLIC

	(*--------------------------------------------------*)
	(* RESET of alarms and warnings 					*)
	(*--------------------------------------------------*)
	xTON_200msTick(IN:= NOT xTON_200msTick.Q, PT:= T#180ms);							(* 180ms + 2x cycle time = 200 ms *)

	IF xTON_200msTick.Q THEN															(* to notice the alarm in 100ms Task *)
	    bAMM_Pr_Ch_P1LP_A_Ms	:= FALSE;
	    bAMM_Pr_Ch_P1LP_B_Ms	:= FALSE;

		bAMM_Pr_Ch_P2LP_Ms		:= FALSE;
		bAMM_Pr_Ch_P2LP_A_Ms	:= FALSE;
	    bAMM_Pr_Ch_P2LP_B_Ms	:= FALSE;

		bAMM_Pr_Ch_P1HP_Ms		:= FALSE;
		bAMM_Pr_Ch_P1HP_A_Ms	:= FALSE;
		bAMM_Pr_Ch_P1HP_B_Ms	:= FALSE;

		bAMM_Pr_Ch_P2HP_Ms		:= FALSE;
		bAMM_Pr_Ch_P2HP_A_Ms	:= FALSE;
		bAMM_Pr_Ch_P2HP_B_Ms	:= FALSE;

	    bAMM_Pr_Ch_P2bFA_Ms		:= FALSE;

		bAMM_Pr_Ch_P2_MsMs		:= FALSE;
		bAMM_Pr_Ch_P2_A_Ms		:= FALSE;
		bAMM_Pr_Ch_P2_B_Ms		:= FALSE;
		bAMM_Pr_Ch_P2_Sum_MsMs	:= FALSE;

		bAMM_Pr_Ch_P2s_MsMs		:= FALSE;
		bAMM_Pr_Ch_P2s_A_Ms		:= FALSE;
		bAMM_Pr_Ch_P2s_B_Ms		:= FALSE;

		bAMM_DPr_Ch_P2_Hi		:= FALSE;
		bAMM_DPr_Ch_P2s_Hi		:= FALSE;
		bAMM_DPr_Ch_P2s_HiHi	:= FALSE;

		bAMM_DPr_Ch_LPCooler_Hi	:= FALSE;
		bAMM_DPr_Ch_HPCooler_Hi	:= FALSE;
		bAMM_DPr_Ch_FA_Hi		:= FALSE;
	END_IF

	OUT_CH.bAMM_Pr_Ch_P2s_Avg	:= FALSE;								(* collective warning *)
	OUT_CH.bAMM_Pr_Ch_P2_Avg	:= FALSE;
	OUT_CH.bAMM_Pr_Ch_P2HP_Avg	:= FALSE;
	OUT_CH.bAMM_Pr_Ch_P1HP_Avg	:= FALSE;
	OUT_CH.bAMM_Pr_Ch_P2LP_Avg	:= FALSE;
	OUT_CH.bAMM_Pr_Ch_P1LP_Avg	:= FALSE;

	(*--------------------------------------------------*)
	(* VISU var of module 								*)
	(*--------------------------------------------------*)
	MM2VIS.rPr_Ch_P1LP_A		:= IN_CH.tPr_Ch_P1LP_A.Ai;
	MM2VIS.rPr_Ch_P1LP_B		:= IN_CH.tPr_Ch_P1LP_B.Ai;

	MM2VIS.rPr_Ch_P2LP      	:= IN_CH.tPr_Ch_P2LP.Ai;
	MM2VIS.rPr_Ch_P2LP_A      	:= IN_CH.tPr_Ch_P2LP_A.Ai;
	MM2VIS.rPr_Ch_P2LP_B      	:= IN_CH.tPr_Ch_P2LP_B.Ai;

	MM2VIS.rPr_Ch_P1HP			:= IN_CH.tPr_Ch_P1HP.Ai;
	MM2VIS.rPr_Ch_P1HP_A		:= IN_CH.tPr_Ch_P1HP_A.Ai;
	MM2VIS.rPr_Ch_P1HP_B		:= IN_CH.tPr_Ch_P1HP_B.Ai;

	MM2VIS.rPr_Ch_P2HP			:= IN_CH.tPr_Ch_P2HP.Ai;
	MM2VIS.rPr_Ch_P2HP_A		:= IN_CH.tPr_Ch_P2HP_A.Ai;
	MM2VIS.rPr_Ch_P2HP_B		:= IN_CH.tPr_Ch_P2HP_B.Ai;

	MM2VIS.rPr_Ch_P2bFA			:= IN_CH.tPr_Ch_P2bFA.Ai;

	MM2VIS.rPr_Ch_P2			:= IN_CH.tPr_Ch_P2.Ai;
	MM2VIS.rPr_Ch_P2_A			:= IN_CH.tPr_Ch_P2_A.Ai;
	MM2VIS.rPr_Ch_P2_B			:= IN_CH.tPr_Ch_P2_B.Ai;

	MM2VIS.rPr_Ch_P2s			:= IN_CH.tPr_Ch_P2s.Ai;
	MM2VIS.rPr_Ch_P2s_A			:= IN_CH.tPr_Ch_P2s_A.Ai;
	MM2VIS.rPr_Ch_P2s_B			:= IN_CH.tPr_Ch_P2s_B.Ai;
	MM2VIS.rPr_Ch_P2s_UF		:= IN_CH.tPr_Ch_P2s.Unfilt;				(* Only for trending *)
	MM2VIS.rPr_Ch_P2s_A_UF		:= IN_CH.tPr_Ch_P2s_A.Unfilt;			(* Only for trending *)
	MM2VIS.rPr_Ch_P2s_B_UF		:= IN_CH.tPr_Ch_P2s_B.Unfilt;			(* Only for trending *)

	MM2VIS.rDPr_Ch_LPCooler		:= 0;
	MM2VIS.rDPr_Ch_HPCooler		:= 0;
	MM2VIS.rDPr_Ch_FA			:= 0;

	(*------------------------------------------------------------------------------------------------------------------------------*)
	(* release for error monitoring 																								*)
	(*------------------------------------------------------------------------------------------------------------------------------*)
	IF bRelModul_ParaSetupOk AND IN_CH.tPB2MM.bSys_Run THEN

		(*----------------------------------------------*)
		(* measurement signal failure 					*)
		(*----------------------------------------------*)
		(* charge pressure p1 before low pressure TC *)
		bAMM_Pr_Ch_P1LP_A_Ms		:= Para.bPr_Ch_P1LP_A_Exist	AND NOT IN_CH.tPr_Ch_P1LP_A.GoodQual;						(* W2779 *)
		bAMM_Pr_Ch_P1LP_B_Ms		:= Para.bPr_Ch_P1LP_B_Exist	AND NOT IN_CH.tPr_Ch_P1LP_B.GoodQual;						(* W2780 *)

			(* release monitoring - delayed reswitch to valid meas.value *)
			xTON_RelMon_P1LP_A(IN	:= Para.bPr_Ch_P1LP_A_Exist AND NOT bAMM_Pr_Ch_P1LP_A_Ms, 	PT:= T#10s);
			xTON_RelMon_P1LP_B(IN	:= Para.bPr_Ch_P1LP_B_Exist AND NOT bAMM_Pr_Ch_P1LP_B_Ms, 	PT:= T#10s);
			bRelMon_P1LP_A			:= xTON_RelMon_P1LP_A.Q;
			bRelMon_P1LP_B			:= xTON_RelMon_P1LP_B.Q;

		(* charge pressure p2 after low pressure TC *)
	    bAMM_Pr_Ch_P2LP_Ms			:= Para.bPr_Ch_P2LP_Exist  	AND NOT IN_CH.tPr_Ch_P2LP.GoodQual;							(* W2668 *)
	    bAMM_Pr_Ch_P2LP_A_Ms		:= Para.bPr_Ch_P2LP_A_Exist AND NOT IN_CH.tPr_Ch_P2LP_A.GoodQual;						(* W2409 *)
	    bAMM_Pr_Ch_P2LP_B_Ms		:= Para.bPr_Ch_P2LP_B_Exist AND NOT IN_CH.tPr_Ch_P2LP_B.GoodQual;						(* W2410 *)

			(* release monitoring - delayed reswitch to valid meas.value *)
			xTON_RelMon_P2LP(IN		:= Para.bPr_Ch_P2LP_Exist   AND NOT bAMM_Pr_Ch_P2LP_Ms,  	PT:= T#10s);
			xTON_RelMon_P2LP_A(IN	:= Para.bPr_Ch_P2LP_A_Exist AND NOT bAMM_Pr_Ch_P2LP_A_Ms, 	PT:= T#10s);
			xTON_RelMon_P2LP_B(IN	:= Para.bPr_Ch_P2LP_B_Exist AND NOT bAMM_Pr_Ch_P2LP_B_Ms, 	PT:= T#10s);
			bRelMon_P2LP			:= xTON_RelMon_P2LP.Q;
			bRelMon_P2LP_A			:= xTON_RelMon_P2LP_A.Q;
			bRelMon_P2LP_B			:= xTON_RelMon_P2LP_B.Q;

		(* charge pressure p1 before high pressure TC *)
		bAMM_Pr_Ch_P1HP_Ms	 		:= Para.bPr_Ch_P1HP_Exist	AND NOT IN_CH.tPr_Ch_P1HP.GoodQual;				(* W2618 *)	(* W9240 *)
		bAMM_Pr_Ch_P1HP_A_Ms		:= Para.bPr_Ch_P1HP_A_Exist	AND NOT IN_CH.tPr_Ch_P1HP_A.GoodQual;			(* W2611 *)	(* W9241 *)
		bAMM_Pr_Ch_P1HP_B_Ms 		:= Para.bPr_Ch_P1HP_B_Exist	AND NOT IN_CH.tPr_Ch_P1HP_B.GoodQual;			(* W2612 *)	(* W9242 *)

			(* release monitoring - delayed reswitch to valid meas.value *)
			xTON_RelMon_P1HP(IN		:= Para.bPr_Ch_P1HP_Exist   AND NOT bAMM_Pr_Ch_P1HP_Ms,  	PT:= T#10s);
			xTON_RelMon_P1HP_A(IN	:= Para.bPr_Ch_P1HP_A_Exist AND NOT bAMM_Pr_Ch_P1HP_A_Ms, 	PT:= T#10s);
			xTON_RelMon_P1HP_B(IN	:= Para.bPr_Ch_P1HP_B_Exist AND NOT bAMM_Pr_Ch_P1HP_B_Ms, 	PT:= T#10s);
			bRelMon_P1HP			:= xTON_RelMon_P1HP.Q;
			bRelMon_P1HP_A			:= xTON_RelMon_P1HP_A.Q;
			bRelMon_P1HP_B			:= xTON_RelMon_P1HP_B.Q;

		(* charge pressure p2 after high pressure TC *)
	    bAMM_Pr_Ch_P2HP_Ms			:= Para.bPr_Ch_P2HP_Exist  	AND NOT IN_CH.tPr_Ch_P2HP.GoodQual;				(* W2669 *)	(* W9237 *)
	    bAMM_Pr_Ch_P2HP_A_Ms		:= Para.bPr_Ch_P2HP_A_Exist AND NOT IN_CH.tPr_Ch_P2HP_A.GoodQual;			(* W2407 *)	(* W9238 *)
	    bAMM_Pr_Ch_P2HP_B_Ms		:= Para.bPr_Ch_P2HP_B_Exist AND NOT IN_CH.tPr_Ch_P2HP_B.GoodQual;			(* W2408 *)	(* W9239 *)

			(* release monitoring - delayed reswitch to valid meas.value *)
			xTON_RelMon_P2HP(IN		:= Para.bPr_Ch_P2HP_Exist   AND NOT bAMM_Pr_Ch_P2HP_Ms,  	PT:= T#10s);
			xTON_RelMon_P2HP_A(IN	:= Para.bPr_Ch_P2HP_A_Exist AND NOT bAMM_Pr_Ch_P2HP_A_Ms, 	PT:= T#10s);
			xTON_RelMon_P2HP_B(IN	:= Para.bPr_Ch_P2HP_B_Exist AND NOT bAMM_Pr_Ch_P2HP_B_Ms, 	PT:= T#10s);
			bRelMon_P2HP			:= xTON_RelMon_P2HP.Q;
			bRelMon_P2HP_A			:= xTON_RelMon_P2HP_A.Q;
			bRelMon_P2HP_B			:= xTON_RelMon_P2HP_B.Q;

		(* charge pressure p2 before flame arrester *)
	    bAMM_Pr_Ch_P2bFA_Ms			:= Para.bPr_Ch_P2bFA_Exist 	AND NOT IN_CH.tPr_Ch_P2bFA.GoodQual;						(* W2670 *)

			(* release monitoring - delayed reswitch to valid meas.value *)
			xTON_RelMon_P2bFA(IN	:= Para.bPr_Ch_P2bFA_Exist	AND NOT bAMM_Pr_Ch_P2bFA_Ms,  	PT:= T#10s);
			bRelMon_P2bFA			:= xTON_RelMon_P2bFA.Q;

		(* charge pressure p2 *)
		bAMM_Pr_Ch_P2_MsMs 			:= Para.bPr_Ch_P2_Exist		AND NOT IN_CH.tPr_Ch_P2.GoodQual;							(* A1077 *)
		bAMM_Pr_Ch_P2_A_Ms 			:= Para.bPr_Ch_P2_A_Exist	AND NOT IN_CH.tPr_Ch_P2_A.GoodQual;							(* W2541 *)
		bAMM_Pr_Ch_P2_B_Ms			:= Para.bPr_Ch_P2_B_Exist	AND NOT IN_CH.tPr_Ch_P2_B.GoodQual;							(* W2543 *)

			(* release monitoring - delayed reswitch to valid meas.value *)
			xTON_RelMon_P2(IN		:= Para.bPr_Ch_P2_Exist   	AND NOT bAMM_Pr_Ch_P2_MsMs,  	PT:= T#10s);
			xTON_RelMon_P2_A(IN		:= Para.bPr_Ch_P2_A_Exist 	AND NOT bAMM_Pr_Ch_P2_A_Ms, 	PT:= T#10s);
			xTON_RelMon_P2_B(IN		:= Para.bPr_Ch_P2_B_Exist 	AND NOT bAMM_Pr_Ch_P2_B_Ms, 	PT:= T#10s);
			bRelMon_P2				:= xTON_RelMon_P2.Q;
			bRelMon_P2_A			:= xTON_RelMon_P2_A.Q;
			bRelMon_P2_B			:= xTON_RelMon_P2_B.Q;

		(* charge pressure p2' *)
		bAMM_Pr_Ch_P2s_MsMs 		:= Para.bPr_Ch_P2s_Exist	AND NOT IN_CH.tPr_Ch_P2s.GoodQual;							(* A1078 *)
		bAMM_Pr_Ch_P2s_A_Ms 		:= Para.bPr_Ch_P2s_A_Exist	AND NOT IN_CH.tPr_Ch_P2s_A.GoodQual;						(* W2539 *)
		bAMM_Pr_Ch_P2s_B_Ms 		:= Para.bPr_Ch_P2s_B_Exist	AND NOT IN_CH.tPr_Ch_P2s_B.GoodQual;						(* W2540 *)

			(* release monitoring	*)
			xTON_RelMon_P2s(IN		:= Para.bPr_Ch_P2s_Exist   	AND NOT bAMM_Pr_Ch_P2s_MsMs,  	PT:= T#10s);
			xTON_RelMon_P2s_A(IN	:= Para.bPr_Ch_P2s_A_Exist 	AND NOT bAMM_Pr_Ch_P2s_A_Ms, 	PT:= T#10s);
			xTON_RelMon_P2s_B(IN	:= Para.bPr_Ch_P2s_B_Exist 	AND NOT bAMM_Pr_Ch_P2s_B_Ms, 	PT:= T#10s);
			bRelMon_P2s				:= xTON_RelMon_P2s.Q;
			bRelMon_P2s_A			:= xTON_RelMon_P2s_A.Q;
			bRelMon_P2s_B			:= xTON_RelMon_P2s_B.Q;

		(* sum failure after a time delay of 48 hours in case of p2 or p2' measuring failure *)
		xTON_ErrMs(IN 				:= bAMM_Pr_Ch_P2s_A_Ms OR bAMM_Pr_Ch_P2s_B_Ms OR bAMM_Pr_Ch_P2_A_Ms OR bAMM_Pr_Ch_P2_B_Ms,
				   PT 				:= T#48h);

		bAMM_Pr_Ch_P2_Sum_MsMs  	:= (xTON_ErrMs.Q AND NOT xEngType.Type9) OR												(* A1078 *)
									   (* measuring failure at all p2 and p2' sensors *)
									   ((bAMM_Pr_Ch_P2s_MsMs   	OR NOT Para.bPr_Ch_P2s_Exist)	AND
										(bAMM_Pr_Ch_P2s_A_Ms 	OR NOT Para.bPr_Ch_P2s_A_Exist) AND
										(bAMM_Pr_Ch_P2s_B_Ms 	OR NOT Para.bPr_Ch_P2s_B_Exist) AND
										(bAMM_Pr_Ch_P2_MsMs		OR NOT Para.bPr_Ch_P2_Exist)	AND
										(bAMM_Pr_Ch_P2_A_Ms  	OR NOT Para.bPr_Ch_P2_A_Exist)  AND
										(bAMM_Pr_Ch_P2_B_Ms		OR NOT Para.bPr_Ch_P2_B_Exist)	   );

		(*----------------------------------------------*)
		(* charge pressure deviation (Spreizung)		*)
		(*----------------------------------------------*)
		bDPr_P2_Hi			:= (ABS(IN_CH.tPr_Ch_P2_A.Ai  - IN_CH.tPr_Ch_P2_B.Ai)  > Para.rPr_Ch_P2s_Diff_HiHi)	AND
							   	bRelMon_P2_A							   	 									AND
								bRelMon_P2_B;

		bDPr_P2s_Hi			:= (ABS(IN_CH.tPr_Ch_P2s_A.Ai - IN_CH.tPr_Ch_P2s_B.Ai) > Para.rPr_Ch_P2s_Diff_HiHi) AND
							    bRelMon_P2s_A 						     										AND
								bRelMon_P2s_B;

		IF bP_Nom10_60s THEN
			bAMM_DPr_Ch_P2_Hi		:=  bDPr_P2_Hi;																			(* W2530 *)
			bAMM_DPr_Ch_P2s_Hi		:= (bDPr_P2s_Hi AND 	xEngType.Type9);												(* W2530 *)
			bAMM_DPr_Ch_P2s_HiHi	:= (bDPr_P2s_Hi AND NOT xEngType.Type9) OR 												(* A2236 *)
									   (bDPr_P2_Hi  AND (bAMM_Pr_Ch_P2s_A_Ms OR bAMM_Pr_Ch_P2s_B_Ms));
		END_IF

		(*--------------------------------------------------------------------------------------------------------------------------*)
		(* Handover charge pressure to other modules																				*)
		(*--------------------------------------------------------------------------------------------------------------------------*)
		(* charge pressure p2' *)
		IF 		bRelMon_P2s 		 THEN 	OUT_CH.rPr_Ch_P2s_Avg 		:= IN_CH.tPr_Ch_P2s.Ai;
											OUT_CH.rPr_Ch_P2s_Max		:= IN_CH.tPr_Ch_P2s.Ai;
											OUT_CH.rPr_Ch_P2s_A 		:= 0;
											OUT_CH.rPr_Ch_P2s_B 		:= 0;
											OUT_CH.rPr_Ch_P2s_Avg_UF 	:= IN_CH.tPr_Ch_P2s.Unfilt;
											OUT_CH.rPr_Ch_P2s_A_UF 		:= 0;
											OUT_CH.rPr_Ch_P2s_B_UF 		:= 0;
		ELSE
			IF 	bRelMon_P2s_A 	 	THEN
				IF bRelMon_P2s_B 	THEN	OUT_CH.rPr_Ch_P2s_Avg		:=(IN_CH.tPr_Ch_P2s_A.Ai + IN_CH.tPr_Ch_P2s_B.Ai) / 2;
											OUT_CH.rPr_Ch_P2s_Max		:= MAX(IN_CH.tPr_Ch_P2s_A.Ai, IN_CH.tPr_Ch_P2s_B.Ai);
											OUT_CH.rPr_Ch_P2s_A 		:= IN_CH.tPr_Ch_P2s_A.Ai;
											OUT_CH.rPr_Ch_P2s_B 		:= IN_CH.tPr_Ch_P2s_B.Ai;
											OUT_CH.rPr_Ch_P2s_Avg_UF	:=(IN_CH.tPr_Ch_P2s_A.Unfilt + IN_CH.tPr_Ch_P2s_B.Unfilt) /2;
											OUT_CH.rPr_Ch_P2s_A_UF 		:= IN_CH.tPr_Ch_P2s_A.Unfilt;
											OUT_CH.rPr_Ch_P2s_B_UF 		:= IN_CH.tPr_Ch_P2s_B.Unfilt;
									ELSE	OUT_CH.rPr_Ch_P2s_Avg 		:= IN_CH.tPr_Ch_P2s_A.Ai;
											OUT_CH.rPr_Ch_P2s_Max		:= IN_CH.tPr_Ch_P2s_A.Ai;
											OUT_CH.rPr_Ch_P2s_A 		:= IN_CH.tPr_Ch_P2s_A.Ai;
											OUT_CH.rPr_Ch_P2s_B 		:= IN_CH.tPr_Ch_P2s_A.Ai;
											OUT_CH.rPr_Ch_P2s_Avg_UF 	:= IN_CH.tPr_Ch_P2s_A.Unfilt;
											OUT_CH.rPr_Ch_P2s_A_UF 		:= IN_CH.tPr_Ch_P2s_A.Unfilt;
											OUT_CH.rPr_Ch_P2s_B_UF 		:= IN_CH.tPr_Ch_P2s_A.Unfilt;
				END_IF
			ELSE
				IF bRelMon_P2s_B 	THEN	OUT_CH.rPr_Ch_P2s_Avg 		:= IN_CH.tPr_Ch_P2s_B.Ai;
											OUT_CH.rPr_Ch_P2s_Max		:= IN_CH.tPr_Ch_P2s_B.Ai;
											OUT_CH.rPr_Ch_P2s_A 		:= IN_CH.tPr_Ch_P2s_B.Ai;
											OUT_CH.rPr_Ch_P2s_B 		:= IN_CH.tPr_Ch_P2s_B.Ai;
											OUT_CH.rPr_Ch_P2s_Avg_UF 	:= IN_CH.tPr_Ch_P2s_B.Unfilt;
											OUT_CH.rPr_Ch_P2s_A_UF 		:= IN_CH.tPr_Ch_P2s_B.Unfilt;
											OUT_CH.rPr_Ch_P2s_B_UF 		:= IN_CH.tPr_Ch_P2s_B.Unfilt;
									ELSE	OUT_CH.rPr_Ch_P2s_Avg 		:= 0;
											OUT_CH.rPr_Ch_P2s_Max		:= 0;
											OUT_CH.rPr_Ch_P2s_A 		:= 0;
											OUT_CH.rPr_Ch_P2s_B 		:= 0;
											OUT_CH.rPr_Ch_P2s_Avg_UF 	:= 0;
											OUT_CH.rPr_Ch_P2s_A_UF 		:= 0;
											OUT_CH.rPr_Ch_P2s_B_UF 		:= 0;
											OUT_CH.bAMM_Pr_Ch_P2s_Avg	:= TRUE;
				END_IF
			END_IF
		END_IF

		MM2VIS.rPr_Ch_P2s_Avg	:= OUT_CH.rPr_Ch_P2s_Avg;					(* VISU *)

		(* charge pressure p2 *)
		IF 		bRelMon_P2 	 		THEN 	OUT_CH.rPr_Ch_P2_Avg 		:= IN_CH.tPr_Ch_P2.Ai;
											OUT_CH.rPr_Ch_P2_Max		:= IN_CH.tPr_Ch_P2.Ai;
		ELSE
			IF 	bRelMon_P2_A 		THEN
				IF bRelMon_P2_B		THEN	OUT_CH.rPr_Ch_P2_Avg		:=(IN_CH.tPr_Ch_P2_A.Ai + IN_CH.tPr_Ch_P2_B.Ai) / 2;
											OUT_CH.rPr_Ch_P2_Max		:= MAX(IN_CH.tPr_Ch_P2_A.Ai, IN_CH.tPr_Ch_P2_B.Ai);
							 		ELSE	OUT_CH.rPr_Ch_P2_Avg 		:= IN_CH.tPr_Ch_P2_A.Ai;
											OUT_CH.rPr_Ch_P2_Max		:= IN_CH.tPr_Ch_P2_A.Ai;
				END_IF
			ELSE
				IF bRelMon_P2_B 	THEN	OUT_CH.rPr_Ch_P2_Avg 		:= IN_CH.tPr_Ch_P2_B.Ai;
											OUT_CH.rPr_Ch_P2_Max		:= IN_CH.tPr_Ch_P2_B.Ai;
									ELSE	OUT_CH.rPr_Ch_P2_Avg 		:= 0;
											OUT_CH.rPr_Ch_P2_Max		:= 0;
											OUT_CH.bAMM_Pr_Ch_P2_Avg	:= TRUE;
				END_IF
			END_IF
		END_IF

		MM2VIS.rPr_Ch_P2_Avg	:= OUT_CH.rPr_Ch_P2_Avg;					(* VISU *)

		(* charge pressure after high-pressure TC *)
		IF 		bRelMon_P2HP 	 	THEN 	OUT_CH.rPr_Ch_P2HP_Avg 		:= IN_CH.tPr_Ch_P2HP.Ai;
											OUT_CH.rPr_Ch_P2HP_Max		:= IN_CH.tPr_Ch_P2HP.Ai;
		ELSE
			IF 	bRelMon_P2HP_A 		THEN
				IF bRelMon_P2HP_B	THEN	OUT_CH.rPr_Ch_P2HP_Avg		:=(IN_CH.tPr_Ch_P2HP_A.Ai + IN_CH.tPr_Ch_P2HP_B.Ai) / 2;
											OUT_CH.rPr_Ch_P2HP_Max		:= MAX(IN_CH.tPr_Ch_P2HP_A.Ai, IN_CH.tPr_Ch_P2HP_B.Ai);
							 		ELSE	OUT_CH.rPr_Ch_P2HP_Avg 		:= IN_CH.tPr_Ch_P2HP_A.Ai;
											OUT_CH.rPr_Ch_P2HP_Max		:= IN_CH.tPr_Ch_P2HP_A.Ai;
				END_IF
			ELSE
				IF bRelMon_P2HP_B 	THEN	OUT_CH.rPr_Ch_P2HP_Avg 		:= IN_CH.tPr_Ch_P2HP_B.Ai;
											OUT_CH.rPr_Ch_P2HP_Max		:= IN_CH.tPr_Ch_P2HP_B.Ai;
									ELSE	OUT_CH.rPr_Ch_P2HP_Avg 		:= 0;
											OUT_CH.rPr_Ch_P2HP_Max		:= 0;
											OUT_CH.bAMM_Pr_Ch_P2HP_Avg	:= TRUE;
				END_IF
			END_IF
		END_IF

		MM2VIS.rPr_Ch_P2HP_Avg	:= OUT_CH.rPr_Ch_P2HP_Avg;					(* VISU *)

		(* charge pressure before high-pressure TC *)
		IF 		bRelMon_P1HP 	 	THEN 	OUT_CH.rPr_Ch_P1HP_Avg 		:= IN_CH.tPr_Ch_P1HP.Ai;
											OUT_CH.rPr_Ch_P1HP_Max		:= IN_CH.tPr_Ch_P1HP.Ai;
		ELSE
			IF 	bRelMon_P1HP_A 		THEN
				IF bRelMon_P1HP_B	THEN	OUT_CH.rPr_Ch_P1HP_Avg		:=(IN_CH.tPr_Ch_P1HP_A.Ai + IN_CH.tPr_Ch_P1HP_B.Ai) / 2;
											OUT_CH.rPr_Ch_P1HP_Max		:= MAX(IN_CH.tPr_Ch_P1HP_A.Ai, IN_CH.tPr_Ch_P1HP_B.Ai);
							 		ELSE	OUT_CH.rPr_Ch_P1HP_Avg 		:= IN_CH.tPr_Ch_P1HP_A.Ai;
											OUT_CH.rPr_Ch_P1HP_Max		:= IN_CH.tPr_Ch_P1HP_A.Ai;
				END_IF
			ELSE
				IF bRelMon_P1HP_B 	THEN	OUT_CH.rPr_Ch_P1HP_Avg 		:= IN_CH.tPr_Ch_P1HP_B.Ai;
											OUT_CH.rPr_Ch_P1HP_Max		:= IN_CH.tPr_Ch_P1HP_B.Ai;
									ELSE	OUT_CH.rPr_Ch_P1HP_Avg 		:= 0;
											OUT_CH.rPr_Ch_P1HP_Max		:= 0;
											OUT_CH.bAMM_Pr_Ch_P1HP_Avg	:= TRUE;
				END_IF
			END_IF
		END_IF

		MM2VIS.rPr_Ch_P1HP_Avg	:= OUT_CH.rPr_Ch_P1HP_Avg;					(* VISU *)

		(* charge pressure after low-pressure TC *)
		IF 		bRelMon_P2LP 	 	THEN 	OUT_CH.rPr_Ch_P2LP_Avg		:= IN_CH.tPr_Ch_P2LP.Ai;
											OUT_CH.rPr_Ch_P2LP_Max		:= IN_CH.tPr_Ch_P2LP.Ai;
		ELSE
			IF 	bRelMon_P2LP_A 	 	THEN
				IF bRelMon_P2LP_B 	THEN	OUT_CH.rPr_Ch_P2LP_Avg		:=(IN_CH.tPr_Ch_P2LP_A.Ai + IN_CH.tPr_Ch_P2LP_B.Ai) / 2;
											OUT_CH.rPr_Ch_P2LP_Max		:= MAX(IN_CH.tPr_Ch_P2LP_A.Ai, IN_CH.tPr_Ch_P2LP_B.Ai);
								 	ELSE	OUT_CH.rPr_Ch_P2LP_Avg 		:= IN_CH.tPr_Ch_P2LP_A.Ai;
											OUT_CH.rPr_Ch_P2LP_Max		:= IN_CH.tPr_Ch_P2LP_A.Ai;
				END_IF
			ELSE
				IF bRelMon_P2LP_B 	THEN	OUT_CH.rPr_Ch_P2LP_Avg 		:= IN_CH.tPr_Ch_P2LP_B.Ai;
											OUT_CH.rPr_Ch_P2LP_Max		:= IN_CH.tPr_Ch_P2LP_B.Ai;
								 	ELSE	OUT_CH.rPr_Ch_P2LP_Avg 		:= 0;
											OUT_CH.rPr_Ch_P2LP_Max		:= 0;
											OUT_CH.bAMM_Pr_Ch_P2LP_Avg	:= TRUE;
				END_IF
			END_IF
		END_IF

		MM2VIS.rPr_Ch_P2LP_Avg	:= OUT_CH.rPr_Ch_P2LP_Avg;					(* VISU *)

		(*charge pressure before low-pressure TC *)
		IF 		bRelMon_P1LP_A 		THEN
			IF 	bRelMon_P1LP_B		THEN	OUT_CH.rPr_Ch_P1LP_Avg		:=(IN_CH.tPr_Ch_P1LP_A.Ai + IN_CH.tPr_Ch_P1LP_B.Ai) / 2;
											OUT_CH.rPr_Ch_P1LP_Max		:= MAX(IN_CH.tPr_Ch_P1LP_A.Ai, IN_CH.tPr_Ch_P1LP_B.Ai);
									ELSE	OUT_CH.rPr_Ch_P1LP_Avg 		:= IN_CH.tPr_Ch_P1LP_A.Ai;
											OUT_CH.rPr_Ch_P1LP_Max		:= IN_CH.tPr_Ch_P1LP_A.Ai;
			END_IF
		ELSIF 	bRelMon_P1LP_B		THEN	OUT_CH.rPr_Ch_P1LP_Avg 		:= IN_CH.tPr_Ch_P1LP_B.Ai;
											OUT_CH.rPr_Ch_P1LP_Max		:= IN_CH.tPr_Ch_P1LP_B.Ai;
									ELSE	OUT_CH.rPr_Ch_P1LP_Avg 		:= 0;
											OUT_CH.rPr_Ch_P1LP_Max		:= 0;
											OUT_CH.bAMM_Pr_Ch_P1LP_Avg	:= TRUE;
		END_IF

		MM2VIS.rPr_Ch_P1LP_Avg	:= OUT_CH.rPr_Ch_P1LP_Avg;					(* VISU *)

		(*--------------------------------------------------------------------------------------------------------------------------*)
		(* Difference pressure over cooler and flame arrester																		*)
		(*--------------------------------------------------------------------------------------------------------------------------*)
		IF 	  NOT OUT_CH.bAMM_Pr_Ch_P2LP_Avg AND NOT OUT_CH.bAMM_Pr_Ch_P1HP_Avg
		THEN
			MM2VIS.rDPr_Ch_LPCooler	:=  MM2VIS.rPr_Ch_P2LP_Avg  - MM2VIS.rPr_Ch_P1HP_Avg;
			bAMM_DPr_Ch_LPCooler_Hi	:= (MM2VIS.rDPr_Ch_LPCooler > Para.rDPr_Ch_LPCooler_Hi) AND bOMSS_MAT;					(* W2671 *)
		END_IF

		IF 	  NOT OUT_CH.bAMM_Pr_Ch_P2HP_Avg AND bRelMon_P2bFA
		THEN
			MM2VIS.rDPr_Ch_HPCooler	:=  MM2VIS.rPr_Ch_P2HP_Avg  - MM2VIS.rPr_Ch_P2bFA;
			bAMM_DPr_Ch_HPCooler_Hi	:= (MM2VIS.rDPr_Ch_HPCooler > Para.rDPr_Ch_HPCooler_Hi)	AND bOMSS_MAT;		(* W2672 *)	(* W9243 *)

		ELSIF NOT OUT_CH.bAMM_Pr_Ch_P2HP_Avg AND NOT OUT_CH.bAMM_Pr_Ch_P2_Avg AND NOT Para.bPr_Ch_P2bFA_Exist
		THEN
			MM2VIS.rDPr_Ch_HPCooler	:=  MM2VIS.rPr_Ch_P2HP_Avg  - MM2VIS.rPr_Ch_P2_Avg;
			bAMM_DPr_Ch_HPCooler_Hi	:= (MM2VIS.rDPr_Ch_HPCooler > Para.rDPr_Ch_HPCooler_Hi)	AND bOMSS_MAT;		(* W2672 *)	(* W9243 *)
		END_IF

		IF 	  NOT OUT_CH.bAMM_Pr_Ch_P2_Avg   AND bRelMon_P2bFA
		THEN
			MM2VIS.rDPr_Ch_FA		:=  MM2VIS.rPr_Ch_P2bFA 	- MM2VIS.rPr_Ch_P2_Avg;
			bAMM_DPr_Ch_FA_Hi		:= (MM2VIS.rDPr_Ch_FA	    > Para.rDPr_Ch_FA_Hi) 		AND bOMSS_MAT;					(* W2673 *)
		END_IF

		(*---------------------------------------------------------------------------------------------------------------------------*)
		(* Monitoring pressures in standstill operation -----------------------------------------------------------------------------*)
		(*---------------------------------------------------------------------------------------------------------------------------*)
		tPr_Ch[0].GoodQual	:= IN_CH.tPr_Ch_P2s.GoodQual;
		tPr_Ch[0].ParaExist	:= Para.bPr_Ch_P2s_Exist;
		tPr_Ch[0].Value 	:= IN_CH.tPr_Ch_P2s.Ai;

		tPr_Ch[1].GoodQual	:= IN_CH.tPr_Ch_P2s_A.GoodQual;
		tPr_Ch[1].ParaExist	:= Para.bPr_Ch_P2s_A_Exist;
		tPr_Ch[1].Value 	:= IN_CH.tPr_Ch_P2s_A.Ai;

		tPr_Ch[2].GoodQual	:= IN_CH.tPr_Ch_P2s_B.GoodQual;
		tPr_Ch[2].ParaExist	:= Para.bPr_Ch_P2s_B_Exist;
		tPr_Ch[2].Value		:= IN_CH.tPr_Ch_P2s_B.Ai;

		tPr_Ch[3].GoodQual	:= IN_CH.tPr_Ch_P2.GoodQual;
		tPr_Ch[3].ParaExist	:= Para.bPr_Ch_P2_Exist;
		tPr_Ch[3].Value		:= IN_CH.tPr_Ch_P2.Ai;

		tPr_Ch[4].GoodQual	:= IN_CH.tPr_Ch_P2_A.GoodQual;
		tPr_Ch[4].ParaExist	:= Para.bPr_Ch_P2_A_Exist;
		tPr_Ch[4].Value 	:= IN_CH.tPr_Ch_P2_A.Ai;

		tPr_Ch[5].GoodQual	:= IN_CH.tPr_Ch_P2_B.GoodQual;
		tPr_Ch[5].ParaExist	:= Para.bPr_Ch_P2_B_Exist;
		tPr_Ch[5].Value 	:= IN_CH.tPr_Ch_P2_B.Ai;

		tPr_Ch[6].GoodQual	:= IN_CH.tPr_Ch_P2LP.GoodQual;
		tPr_Ch[6].ParaExist	:= Para.bPr_Ch_P2LP_Exist;
		tPr_Ch[6].Value 	:= IN_CH.tPr_Ch_P2LP.Ai;

		tPr_Ch[7].GoodQual	:= IN_CH.tPr_Ch_P2LP_A.GoodQual;
		tPr_Ch[7].ParaExist	:= Para.bPr_Ch_P2LP_A_Exist;
		tPr_Ch[7].Value 	:= IN_CH.tPr_Ch_P2LP_A.Ai;

		tPr_Ch[8].GoodQual	:= IN_CH.tPr_Ch_P2LP_B.GoodQual;
		tPr_Ch[8].ParaExist	:= Para.bPr_Ch_P2LP_B_Exist;
		tPr_Ch[8].Value 	:= IN_CH.tPr_Ch_P2LP_B.Ai;

		tPr_Ch[9].GoodQual	:= IN_CH.tPr_Ch_P2bFA.GoodQual;
		tPr_Ch[9].ParaExist	:= Para.bPr_Ch_P2bFA_Exist;
		tPr_Ch[9].Value 	:= IN_CH.tPr_Ch_P2bFA.Ai;

		tPr_Ch[10].GoodQual	:= IN_CH.tPr_Ch_P2HP.GoodQual;
		tPr_Ch[10].ParaExist:= Para.bPr_Ch_P2HP_Exist;
		tPr_Ch[10].Value 	:= IN_CH.tPr_Ch_P2HP.Ai;

		tPr_Ch[11].GoodQual	:= IN_CH.tPr_Ch_P2HP_A.GoodQual;
		tPr_Ch[11].ParaExist:= Para.bPr_Ch_P2HP_A_Exist;
		tPr_Ch[11].Value 	:= IN_CH.tPr_Ch_P2HP_A.Ai;

		tPr_Ch[12].GoodQual	:= IN_CH.tPr_Ch_P2HP_B.GoodQual;
		tPr_Ch[12].ParaExist:= Para.bPr_Ch_P2HP_B_Exist;
		tPr_Ch[12].Value 	:= IN_CH.tPr_Ch_P2HP_B.Ai;

		tPr_Ch[13].GoodQual	:= IN_CH.tPr_Ch_P1HP.GoodQual;
		tPr_Ch[13].ParaExist:= Para.bPr_Ch_P1HP_Exist;
		tPr_Ch[13].Value 	:= IN_CH.tPr_Ch_P1HP.Ai;

		tPr_Ch[14].GoodQual	:= IN_CH.tPr_Ch_P1HP_A.GoodQual;
		tPr_Ch[14].ParaExist:= Para.bPr_Ch_P1HP_A_Exist;
		tPr_Ch[14].Value 	:= IN_CH.tPr_Ch_P1HP_A.Ai;

		tPr_Ch[15].GoodQual	:= IN_CH.tPr_Ch_P1HP_B.GoodQual;
		tPr_Ch[15].ParaExist:= Para.bPr_Ch_P1HP_B_Exist;
		tPr_Ch[15].Value 	:= IN_CH.tPr_Ch_P1HP_B.Ai;

		tPr_Ch[16].GoodQual	:= IN_CH.tPr_Ch_P1LP_A.GoodQual;
		tPr_Ch[16].ParaExist:= Para.bPr_Ch_P1LP_A_Exist;
		tPr_Ch[16].Value 	:= IN_CH.tPr_Ch_P1LP_A.Ai;

		tPr_Ch[17].GoodQual	:= IN_CH.tPr_Ch_P1LP_B.GoodQual;
		tPr_Ch[17].ParaExist:= Para.bPr_Ch_P1LP_B_Exist;
		tPr_Ch[17].Value 	:= IN_CH.tPr_Ch_P1LP_B.Ai;

		(* release monitoring charge pressures in standstill *)
		xTON_1sTick(IN := NOT xTON_1sTick.Q, PT:= T#1s);				(* Function executes every 1 second *)

		IF (IN_CH.rN_EngAct = 0) AND (xTON_1sTick.Q) THEN 				(* Engine stopped *)
			iPr_Ch_Out_lgt 	:= 0;
			iPr_Ch_Ok_lgt 	:= 0;

	 		bAMM_Pr_Ch_OoR 	:= FALSE;
			szPr_Ch_OoR		:= '';

			FOR i := 0 TO iPr_Ch_lgt -1 DO								(* For each possible boost pressures *)
				IF  tPr_Ch[i].GoodQual AND tPr_Ch[i].ParaExist THEN		(* Check if it is available *)

			(* First out of range detection *)
					IF tPr_Ch[i].Value < rPr_Ch_Max AND
					   tPr_Ch[i].Value > rPr_Ch_Min
					THEN
						tPr_Ch_Ok[iPr_Ch_Ok_lgt]	:= tPr_Ch[i];
						iPr_Ch_Ok_lgt 				:= iPr_Ch_Ok_lgt + 1;
					ELSE
						tPr_Ch_Out[iPr_Ch_Out_lgt] 	:= tPr_Ch[i];
						iPr_Ch_Out_lgt 				:= iPr_Ch_Out_lgt + 1;
					END_IF
				END_IF
			END_FOR

			(* Start outlier detection method *)
			IF iPr_Ch_Ok_lgt >1 THEN
				FOR i := 1 TO iPr_Ch_Ok_lgt-1 DO						(* Sort pressures from min to max *)
					j := i;
					WHILE (j > 0) DO
						IF (tPr_Ch_Ok[j-1].Value > tPr_Ch_Ok[j].Value) THEN
							tPr_Ch_Tmp 		:= tPr_Ch_Ok[j-1];
							tPr_Ch_Ok[j-1] 	:= tPr_Ch_Ok[j];
							tPr_Ch_Ok[j] 	:= tPr_Ch_Tmp;
							j 				:= j-1;
						ELSE
							EXIT; // End while statement
						END_IF
					END_WHILE
				END_FOR

				IF INT_TO_BOOL(iPr_Ch_Ok_lgt MOD 2) THEN				(* Find median value*)
					rPr_Ch_Ok_medVal := tPr_Ch_Ok[(iPr_Ch_Ok_lgt+1) / 2 - 1].Value;		// odd
				ELSE
					rPr_Ch_Ok_medVal := (tPr_Ch_Ok[iPr_Ch_Ok_lgt / 2 - 1].Value +
										 tPr_Ch_Ok[iPr_Ch_Ok_lgt / 2].Value) / 2;		// even
				END_IF

					iTmp_Pr_Ch_Out_lgt := 0;
					iTmp_Pr_Ch_rest_lgt := 0;

				FOR i := 0 TO iPr_Ch_Ok_lgt-1 DO										(* Tolerance: median +- rPr_Ch_devMax *)
					IF tPr_Ch_Ok[i].Value < (rPr_Ch_Ok_medVal - rPr_Ch_devMax) OR
					   tPr_Ch_Ok[i].Value > (rPr_Ch_Ok_medVal + rPr_Ch_devMax)
					THEN
						tPr_Ch_Out[iPr_Ch_Out_lgt] 	:= tPr_Ch_Ok[i];  					(* Add the values into the outliers array *)
						iPr_Ch_Out_lgt 				:= iPr_Ch_Out_lgt + 1;
						iTmp_Pr_Ch_Out_lgt 			:= iTmp_Pr_Ch_Out_lgt + 1;
					ELSE
						tTmp_Pr_Ch_rest[iTmp_Pr_Ch_rest_lgt] := tPr_Ch_Ok[i];  			(* Add the values into the outliers array *)
						iTmp_Pr_Ch_rest_lgt 		:= iTmp_Pr_Ch_rest_lgt + 1;
					END_IF
				END_FOR
			END_IF

			(* When only 1 value is out, apply outlier detection method in the rest of the array *)
			IF (iTmp_Pr_Ch_Out_lgt = 1) AND (iTmp_Pr_Ch_rest_lgt > 2) THEN
				IF INT_TO_BOOL(iTmp_Pr_Ch_rest_lgt MOD 2) THEN			(* Find median value*)
					rPr_Ch_Ok_medVal := tTmp_Pr_Ch_rest[(iTmp_Pr_Ch_rest_lgt+1)/2 -1].Value;	// odd
				ELSE 																			// even
					rPr_Ch_Ok_medVal := (tTmp_Pr_Ch_rest[iTmp_Pr_Ch_rest_lgt/2 -1].Value
									   + tTmp_Pr_Ch_rest[iTmp_Pr_Ch_rest_lgt/2].Value)/2;
				END_IF

				FOR i := 0 TO iTmp_Pr_Ch_rest_lgt-1 DO										(* Tolerance: median +- rPr_Ch_devMax *)
					IF  tTmp_Pr_Ch_rest[i].Value < (rPr_Ch_Ok_medVal - rPr_Ch_devMax) OR
						tTmp_Pr_Ch_rest[i].Value > (rPr_Ch_Ok_medVal + rPr_Ch_devMax)
					THEN
						tPr_Ch_Out[iPr_Ch_Out_lgt]	:= tPr_Ch_Ok[i];  						(* Add the pressure into the outliers array *)
						iPr_Ch_Out_lgt 				:= iPr_Ch_Out_lgt + 1;
					END_IF
				END_FOR
			END_IF

			(* Warning management *)
			IF iPr_Ch_Out_lgt > 0 THEN
				bAMM_Pr_Ch_OoR 		 := TRUE;

				(* Update associated message *)
				szPr_Ch_OoR := tPr_Ch_Out[0].Tag;
				IF iPr_Ch_Out_lgt > 1 THEN
					FOR i := 1 TO iPr_Ch_Out_lgt-1 DO
						szPr_Ch_OoR := CONCAT(szPr_Ch_OoR, ', ');
						szPr_Ch_OoR := CONCAT(szPr_Ch_OoR, tPr_Ch_Out[i].Tag);
					END_FOR
				END_IF
			END_IF

			MM2VIS.szPr_Ch_OoR 	:= szPr_Ch_OoR;
		END_IF

	ELSE
		xTON_RelMon_P1LP_A(IN	:= FALSE);
		xTON_RelMon_P1LP_B(IN	:= FALSE);
		xTON_RelMon_P2LP(IN		:= FALSE);
		xTON_RelMon_P2LP_A(IN	:= FALSE);
		xTON_RelMon_P2LP_B(IN	:= FALSE);
		xTON_RelMon_P1HP(IN		:= FALSE);
		xTON_RelMon_P1HP_A(IN	:= FALSE);
		xTON_RelMon_P1HP_B(IN	:= FALSE);
		xTON_RelMon_P2HP(IN		:= FALSE);
		xTON_RelMon_P2HP_A(IN	:= FALSE);
		xTON_RelMon_P2HP_B(IN	:= FALSE);
		xTON_RelMon_P2bFA(IN	:= FALSE);
		xTON_RelMon_P2(IN		:= FALSE);
		xTON_RelMon_P2_A(IN		:= FALSE);
		xTON_RelMon_P2_B(IN		:= FALSE);
		xTON_RelMon_P2s(IN		:= FALSE);
		xTON_RelMon_P2s_A(IN	:= FALSE);
		xTON_RelMon_P2s_B(IN	:= FALSE);
		xTON_ErrMs(IN 			:= FALSE);
		xTON_1sTick(IN			:= FALSE);
	END_IF

END_PROGRAM
```
